LIN {X 0,Y 197.942,Z 460.439,A -85,B 0,C 180,E1 -21324.546,E2 -21324.546} C_VEL
LIN {X 0,Y 197.661,Z 463.395,A -85,B 0,C 180,E1 -21327.96,E2 -21327.96} C_VEL
LIN {X 0,Y 197.713,Z 464.596,A -85,B 0,C 180,E1 -21329.998,E2 -21329.998} C_VEL
LIN {X 0,Y 197.549,Z 465.339,A -85,B 0,C 180,E1 -21332.037,E2 -21332.037} C_VEL
LIN {X 0,Y 197.391,Z 465.599,A -85,B 0,C 180,E1 -21336.129,E2 -21336.129} C_VEL
LIN {X 0,Y 197.553,Z 465.155,A -85,B 0,C 180,E1 -21338.179,E2 -21338.179} C_VEL
LIN {X 0,Y 197.931,Z 464.289,A -85,B 0,C 180,E1 -21340.224,E2 -21340.224} C_VEL
LIN {X 0,Y 199.286,Z 461.345,A -85,B 0,C 180,E1 -21344.29,E2 -21344.29} C_VEL
LIN {X 0,Y 201.111,Z 458.021,A -85,B 0,C 180,E1 -21347.278,E2 -21347.278} C_VEL
LIN {X 0,Y 203.402,Z 453.64,A -85,B 0,C 180,E1 -21350.211,E2 -21350.211} C_VEL
LIN {X 0,Y 206.215,Z 447.922,A -85,B 0,C 180,E1 -21353.155,E2 -21353.155} C_VEL
LIN {X 0,Y 209.5,Z 441.158,A -85,B 0,C 180,E1 -21355.853,E2 -21355.853} C_VEL
LIN {X 0,Y 213.512,Z 432.506,A -85,B 0,C 180,E1 -21358.506,E2 -21358.506} C_VEL
LIN {X 0,Y 217.222,Z 423.657,A -85,B 0,C 180,E1 -21360.633,E2 -21360.633} C_VEL
LIN {X 0,Y 220.793,Z 413.95,A -85,B 0,C 180,E1 -21362.487,E2 -21362.487} C_VEL
LIN {X 0,Y 224.184,Z 403.229,A -85,B 0,C 180,E1 -21364.079,E2 -21364.079} C_VEL
LIN {X 0,Y 227.453,Z 391.24,A -85,B 0,C 180,E1 -21365.402,E2 -21365.402} C_VEL
LIN {X 0,Y 230.075,Z 378.731,A -85,B 0,C 180,E1 -21366.421,E2 -21366.421} C_VEL
LIN {X 0,Y 231.955,Z 365.313,A -85,B 0,C 180,E1 -21367.16,E2 -21367.16} C_VEL
LIN {X 0,Y 233.15,Z 348.218,A -85,B 0,C 180,E1 -21367.736,E2 -21367.736} C_VEL
LIN {X 0,Y 234.841,Z 317.353,A -85,B 0,C 180,E1 -21368.645,E2 -21368.645} C_VEL
LIN {X 0,Y 232.576,Z 295.848,A -85,B 0,C 180,E1 -21370.122,E2 -21370.122} C_VEL
LIN {X 0,Y 230.05,Z 288.532,A -85,B 0,C 180,E1 -21371.098,E2 -21371.098} C_VEL
LIN {X 0,Y 224.045,Z 278.534,A -85,B 0,C 180,E1 -21373.235,E2 -21373.235} C_VEL
LIN {X 0,Y 217.477,Z 268.652,A -85,B 0,C 180,E1 -21375.773,E2 -21375.773} C_VEL
LIN {X 0,Y 213.24,Z 263.042,A -85,B 0,C 180,E1 -21377.545,E2 -21377.545} C_VEL
LIN {X 0,Y 210.962,Z 259.841,A -85,B 0,C 180,E1 -21378.571,E2 -21378.571} C_VEL
LIN {X 0,Y 208.26,Z 256.36,A -85,B 0,C 180,E1 -21379.834,E2 -21379.834} C_VEL
LIN {X 0,Y 207.427,Z 255.193,A -85,B 0,C 180,E1 -21380.244,E2 -21380.244} C_VEL
LIN {X 0,Y 204.921,Z 252.53,A -85,B 0,C 180,E1 -21381.473,E2 -21381.473} C_VEL
LIN {X 0,Y 203.6,Z 250.132,A -85,B 0,C 180,E1 -21382.215,E2 -21382.215} C_VEL
LIN {X 0,Y 201.149,Z 248.227,A -85,B 0,C 180,E1 -21383.488,E2 -21383.488} C_VEL
LIN {X 0,Y 199.87,Z 245.754,A -85,B 0,C 180,E1 -21384.296,E2 -21384.296} C_VEL
LIN {X 0,Y 199.655,Z 244.583,A -85,B 0,C 180,E1 -21384.529,E2 -21384.529} C_VEL
LIN {X 0,Y 199.678,Z 244.597,A -85,B 0,C 180,E1 -21388.133,E2 -21388.133} C_VEL
LIN {X 0,Y 199.633,Z 244.592,A -85,B 0,C 180,E1 -21392.764,E2 -21392.764} C_VEL
LIN {X 0,Y 199.67,Z 244.569,A -85,B 0,C 180,E1 -21397.221,E2 -21397.221} C_VEL
LIN {X 0,Y 199.737,Z 244.601,A -85,B 0,C 180,E1 -21401.802,E2 -21401.802} C_VEL
LIN {X 0,Y 199.795,Z 244.552,A -85,B 0,C 180,E1 -21405.746,E2 -21405.746} C_VEL
LIN {X 0,Y 200.015,Z 244.57,A -85,B 0,C 180,E1 -21409.882,E2 -21409.882} C_VEL
LIN {X 0,Y 199.994,Z 244.528,A -85,B 0,C 180,E1 -21413.949,E2 -21413.949} C_VEL
LIN {X 0,Y 200.281,Z 244.53,A -85,B 0,C 180,E1 -21417.99,E2 -21417.99} C_VEL
LIN {X 0,Y 200.44,Z 244.499,A -85,B 0,C 180,E1 -21420,E2 -21420} C_VEL
LIN {X 0,Y 199.992,Z 244.532,A -85,B 0,C 180,E1 -21424.031,E2 -21424.031} C_VEL
LIN {X 0,Y 200.081,Z 244.539,A -85,B 0,C 180,E1 -21428.077,E2 -21428.077} C_VEL
LIN {X 0,Y 199.863,Z 244.559,A -85,B 0,C 180,E1 -21432.181,E2 -21432.181} C_VEL
LIN {X 0,Y 199.782,Z 244.569,A -85,B 0,C 180,E1 -21436.346,E2 -21436.346} C_VEL
LIN {X 0,Y 199.691,Z 244.611,A -85,B 0,C 180,E1 -21440.607,E2 -21440.607} C_VEL
LIN {X 0,Y 199.718,Z 244.604,A -85,B 0,C 180,E1 -21441.956,E2 -21441.956} C_VEL
LIN {X 0,Y 200.527,Z 247.136,A -85,B 0,C 180,E1 -21442.541,E2 -21442.541} C_VEL
LIN {X 0,Y 202.565,Z 249.424,A -85,B 0,C 180,E1 -21443.668,E2 -21443.668} C_VEL
LIN {X 0,Y 203.976,Z 250.475,A -85,B 0,C 180,E1 -21444.381,E2 -21444.381} C_VEL
LIN {X 0,Y 205.845,Z 253.622,A -85,B 0,C 180,E1 -21445.399,E2 -21445.399} C_VEL
LIN {X 0,Y 208.072,Z 255.817,A -85,B 0,C 180,E1 -21446.461,E2 -21446.461} C_VEL
LIN {X 0,Y 210.626,Z 259.382,A -85,B 0,C 180,E1 -21447.678,E2 -21447.678} C_VEL
LIN {X 0,Y 212.048,Z 261.212,A -85,B 0,C 180,E1 -21448.319,E2 -21448.319} C_VEL
LIN {X 0,Y 215.867,Z 266.452,A -85,B 0,C 180,E1 -21449.971,E2 -21449.971} C_VEL
LIN {X 0,Y 221.051,Z 273.806,A -85,B 0,C 180,E1 -21452.044,E2 -21452.044} C_VEL
LIN {X 0,Y 228.397,Z 285.486,A -85,B 0,C 180,E1 -21454.726,E2 -21454.726} C_VEL
LIN {X 0,Y 235.783,Z 298.796,A -85,B 0,C 180,E1 -21457.196,E2 -21457.196} C_VEL
LIN {X 0,Y 236.31,Z 299.86,A -85,B 0,C 180,E1 -21457.367,E2 -21457.367} C_VEL
LIN {X 0,Y 233.51,Z 345.758,A -85,B 0,C 180,E1 -21458.696,E2 -21458.696} C_VEL
LIN {X 0,Y 232.102,Z 359,A -85,B 0,C 180,E1 -21459.385,E2 -21459.385} C_VEL
LIN {X 0,Y 229.988,Z 371.479,A -85,B 0,C 180,E1 -21460.359,E2 -21460.359} C_VEL
LIN {X 0,Y 227.13,Z 384.146,A -85,B 0,C 180,E1 -21461.716,E2 -21461.716} C_VEL
LIN {X 0,Y 223.756,Z 395.932,A -85,B 0,C 180,E1 -21463.423,E2 -21463.423} C_VEL
LIN {X 0,Y 220.104,Z 406.463,A -85,B 0,C 180,E1 -21465.378,E2 -21465.378} C_VEL
LIN {X 0,Y 216.353,Z 415.831,A -85,B 0,C 180,E1 -21467.624,E2 -21467.624} C_VEL
LIN {X 0,Y 212.904,Z 423.462,A -85,B 0,C 180,E1 -21469.935,E2 -21469.935} C_VEL
LIN {X 0,Y 209.261,Z 430.89,A -85,B 0,C 180,E1 -21472.808,E2 -21472.808} C_VEL
LIN {X 0,Y 206.113,Z 436.751,A -85,B 0,C 180,E1 -21475.766,E2 -21475.766} C_VEL
LIN {X 0,Y 203.456,Z 441.257,A -85,B 0,C 180,E1 -21478.795,E2 -21478.795} C_VEL
LIN {X 0,Y 201.95,Z 443.598,A -85,B 0,C 180,E1 -21480.845,E2 -21480.845} C_VEL
LIN {X 0,Y 200.677,Z 445.486,A -85,B 0,C 180,E1 -21482.92,E2 -21482.92} C_VEL
LIN {X 0,Y 198.945,Z 447.673,A -85,B 0,C 180,E1 -21486.707,E2 -21486.707} C_VEL
LIN {X 0,Y 198.092,Z 448.373,A -85,B 0,C 180,E1 -21489.222,E2 -21489.222} C_VEL
LIN {X 0,Y 197.64,Z 448.461,A -85,B 0,C 180,E1 -21491.337,E2 -21491.337} C_VEL
LIN {X 0,Y 197.323,Z 447.972,A -85,B 0,C 180,E1 -21494.084,E2 -21494.084} C_VEL
LIN {X 0,Y 197.162,Z 446.247,A -85,B 0,C 180,E1 -21497.653,E2 -21497.653} C_VEL
LIN {X 0,Y 197.432,Z 443.697,A -85,B 0,C 180,E1 -21500.785,E2 -21500.785} C_VEL
LIN {X 0,Y 198.046,Z 440.117,A -85,B 0,C 180,E1 -21503.891,E2 -21503.891} C_VEL
LIN {X 0,Y 198.809,Z 435.436,A -85,B 0,C 180,E1 -21506.963,E2 -21506.963} C_VEL
LIN {X 0,Y 199.937,Z 429.504,A -85,B 0,C 180,E1 -21510.002,E2 -21510.002} C_VEL
LIN {X 0,Y 201.503,Z 422.11,A -85,B 0,C 180,E1 -21513.001,E2 -21513.001} C_VEL
LIN {X 0,Y 203.143,Z 414.552,A -85,B 0,C 180,E1 -21515.462,E2 -21515.462} C_VEL
LIN {X 0,Y 205.28,Z 404.301,A -85,B 0,C 180,E1 -21518.121,E2 -21518.121} C_VEL
LIN {X 0,Y 207.44,Z 393.458,A -85,B 0,C 180,E1 -21520.33,E2 -21520.33} C_VEL
LIN {X 0,Y 209.325,Z 382.204,A -85,B 0,C 180,E1 -21522.115,E2 -21522.115} C_VEL
LIN {X 0,Y 210.819,Z 369.938,A -85,B 0,C 180,E1 -21523.62,E2 -21523.62} C_VEL
LIN {X 0,Y 212.169,Z 357.731,A -85,B 0,C 180,E1 -21524.693,E2 -21524.693} C_VEL
LIN {X 0,Y 213.122,Z 344.661,A -85,B 0,C 180,E1 -21525.447,E2 -21525.447} C_VEL
LIN {X 0,Y 215.625,Z 279.151,A -85,B 0,C 180,E1 -21527.583,E2 -21527.583} C_VEL
LIN {X 0,Y 208.838,Z 263.06,A -85,B 0,C 180,E1 -21529.128,E2 -21529.128} C_VEL
LIN {X 0,Y 201.032,Z 247.936,A -85,B 0,C 180,E1 -21530.917,E2 -21530.917} C_VEL
LIN {X 0,Y 199.755,Z 244.973,A -85,B 0,C 180,E1 -21531.246,E2 -21531.246} C_VEL
LIN {X 0,Y 199.699,Z 244.61,A -85,B 0,C 180,E1 -21531.317,E2 -21531.317} C_VEL
LIN {X 0,Y 199.647,Z 244.616,A -85,B 0,C 180,E1 -21534.99,E2 -21534.99} C_VEL
LIN {X 0,Y 199.613,Z 244.619,A -85,B 0,C 180,E1 -21539.535,E2 -21539.535} C_VEL
LIN {X 0,Y 199.671,Z 244.612,A -85,B 0,C 180,E1 -21542.354,E2 -21542.354} C_VEL
LIN {X 0,Y 199.623,Z 244.611,A -85,B 0,C 180,E1 -21546.766,E2 -21546.766} C_VEL
LIN {X 0,Y 199.601,Z 244.623,A -85,B 0,C 180,E1 -21549.333,E2 -21549.333} C_VEL
LIN {X 0,Y 199.572,Z 244.612,A -85,B 0,C 180,E1 -21552.308,E2 -21552.308} C_VEL
LIN {X 0,Y 199.582,Z 244.619,A -85,B 0,C 180,E1 -21555.228,E2 -21555.228} C_VEL
LIN {X 0,Y 199.575,Z 244.621,A -85,B 0,C 180,E1 -21558.003,E2 -21558.003} C_VEL
LIN {X 0,Y 199.602,Z 244.602,A -85,B 0,C 180,E1 -21560.774,E2 -21560.774} C_VEL
LIN {X 0,Y 199.617,Z 244.617,A -85,B 0,C 180,E1 -21565.714,E2 -21565.714} C_VEL
LIN {X 0,Y 199.692,Z 244.605,A -85,B 0,C 180,E1 -21568.135,E2 -21568.135} C_VEL
LIN {X 0,Y 199.734,Z 244.589,A -85,B 0,C 180,E1 -21572.188,E2 -21572.188} C_VEL
LIN {X 0,Y 206.813,Z 272.195,A -85,B 0,C 180,E1 -21574.133,E2 -21574.133} C_VEL
LIN {X 0,Y 203.31,Z 347.013,A -85,B 0,C 180,E1 -21578.76,E2 -21578.76} C_VEL
LIN {X 0,Y 202.562,Z 361.775,A -85,B 0,C 180,E1 -21580.095,E2 -21580.095} C_VEL
LIN {X 0,Y 201.607,Z 374.93,A -85,B 0,C 180,E1 -21581.715,E2 -21581.715} C_VEL
LIN {X 0,Y 200.603,Z 387.656,A -85,B 0,C 180,E1 -21583.723,E2 -21583.723} C_VEL
LIN {X 0,Y 199.784,Z 399.17,A -85,B 0,C 180,E1 -21586.004,E2 -21586.004} C_VEL
LIN {X 0,Y 199.015,Z 408.647,A -85,B 0,C 180,E1 -21588.284,E2 -21588.284} C_VEL
LIN {X 0,Y 198.445,Z 417.441,A -85,B 0,C 180,E1 -21590.829,E2 -21590.829} C_VEL
LIN {X 0,Y 198.005,Z 426.054,A -85,B 0,C 180,E1 -21593.887,E2 -21593.887} C_VEL
LIN {X 0,Y 197.786,Z 433.046,A -85,B 0,C 180,E1 -21596.944,E2 -21596.944} C_VEL
LIN {X 0,Y 197.683,Z 438.659,A -85,B 0,C 180,E1 -21600,E2 -21600} C_VEL
LIN {X 0,Y 197.968,Z 443.125,A -85,B 0,C 180,E1 -21603.052,E2 -21603.052} C_VEL
LIN {X 0,Y 198.708,Z 446.59,A -85,B 0,C 180,E1 -21606.09,E2 -21606.09} C_VEL
LIN {X 0,Y 200.084,Z 449.8,A -85,B 0,C 180,E1 -21610.115,E2 -21610.115} C_VEL
LIN {X 0,Y 201.178,Z 450.837,A -85,B 0,C 180,E1 -21612.099,E2 -21612.099} C_VEL
LIN {X 0,Y 204.584,Z 451.772,A -85,B 0,C 180,E1 -21615.951,E2 -21615.951} C_VEL
LIN {X 0,Y 208.896,Z 451.263,A -85,B 0,C 180,E1 -21619.659,E2 -21619.659} C_VEL
LIN {X 0,Y 214.052,Z 449.305,A -85,B 0,C 180,E1 -21623.203,E2 -21623.203} C_VEL
LIN {X 0,Y 220.272,Z 445.773,A -85,B 0,C 180,E1 -21626.531,E2 -21626.531} C_VEL
LIN {X 0,Y 224.069,Z 443.144,A -85,B 0,C 180,E1 -21628.292,E2 -21628.292} C_VEL
LIN {X 0,Y 226.413,Z 441.172,A -85,B 0,C 180,E1 -21629.578,E2 -21629.578} C_VEL
LIN {X 0,Y 231.508,Z 435.44,A -85,B 0,C 180,E1 -21633.602,E2 -21633.602} C_VEL
LIN {X 0,Y 233.945,Z 432.914,A -85,B 0,C 180,E1 -21634.759,E2 -21634.759} C_VEL
LIN {X 0,Y 234.952,Z 431.935,A -85,B 0,C 180,E1 -21635.093,E2 -21635.093} C_VEL
LIN {X 0,Y 243.29,Z 423.495,A -85,B 0,C 180,E1 -21637.346,E2 -21637.346} C_VEL
LIN {X 0,Y 250.623,Z 414.818,A -85,B 0,C 180,E1 -21639.12,E2 -21639.12} C_VEL
LIN {X 0,Y 258.387,Z 404.268,A -85,B 0,C 180,E1 -21640.752,E2 -21640.752} C_VEL
LIN {X 0,Y 265.576,Z 392.717,A -85,B 0,C 180,E1 -21642.106,E2 -21642.106} C_VEL
LIN {X 0,Y 271.928,Z 380.59,A -85,B 0,C 180,E1 -21643.21,E2 -21643.21} C_VEL
LIN {X 0,Y 276.977,Z 368.919,A -85,B 0,C 180,E1 -21643.996,E2 -21643.996} C_VEL
LIN {X 0,Y 276.871,Z 369.239,A -85,B 0,C 180,E1 -21644.215,E2 -21644.215} C_VEL
LIN {X 0,Y 271.282,Z 382.338,A -85,B 0,C 180,E1 -21644.913,E2 -21644.913} C_VEL
LIN {X 0,Y 264.304,Z 395.717,A -85,B 0,C 180,E1 -21645.885,E2 -21645.885} C_VEL
LIN {X 0,Y 256.722,Z 407.968,A -85,B 0,C 180,E1 -21647.078,E2 -21647.078} C_VEL
LIN {X 0,Y 249.17,Z 418.536,A -85,B 0,C 180,E1 -21648.482,E2 -21648.482} C_VEL
LIN {X 0,Y 241.34,Z 428.187,A -85,B 0,C 180,E1 -21650.157,E2 -21650.157} C_VEL
LIN {X 0,Y 233.944,Z 436.234,A -85,B 0,C 180,E1 -21651.984,E2 -21651.984} C_VEL
LIN {X 0,Y 227.076,Z 442.972,A -85,B 0,C 180,E1 -21653.979,E2 -21653.979} C_VEL
LIN {X 0,Y 218.693,Z 450.246,A -85,B 0,C 180,E1 -21656.883,E2 -21656.883} C_VEL
LIN {X 0,Y 212.811,Z 454.741,A -85,B 0,C 180,E1 -21659.343,E2 -21659.343} C_VEL
LIN {X 0,Y 207.842,Z 458.064,A -85,B 0,C 180,E1 -21661.743,E2 -21661.743} C_VEL
LIN {X 0,Y 202.079,Z 461.387,A -85,B 0,C 180,E1 -21665.331,E2 -21665.331} C_VEL
LIN {X 0,Y 197.481,Z 463.356,A -85,B 0,C 180,E1 -21669.15,E2 -21669.15} C_VEL
LIN {X 0,Y 193.954,Z 463.965,A -85,B 0,C 180,E1 -21673.147,E2 -21673.147} C_VEL
LIN {X 0,Y 191.876,Z 463.198,A -85,B 0,C 180,E1 -21677.302,E2 -21677.302} C_VEL
LIN {X 0,Y 191.007,Z 461.056,A -85,B 0,C 180,E1 -21681.534,E2 -21681.534} C_VEL
LIN {X 0,Y 191.007,Z 459.364,A -85,B 0,C 180,E1 -21683.798,E2 -21683.798} C_VEL
LIN {X 0,Y 190.663,Z 461.301,A -85,B 0,C 180,E1 -21685.77,E2 -21685.77} C_VEL
LIN {X 0,Y 190.578,Z 462.945,A -85,B 0,C 180,E1 -21687.884,E2 -21687.884} C_VEL
LIN {X 0,Y 190.642,Z 464.177,A -85,B 0,C 180,E1 -21689.998,E2 -21689.998} C_VEL
LIN {X 0,Y 190.457,Z 464.976,A -85,B 0,C 180,E1 -21692.112,E2 -21692.112} C_VEL
LIN {X 0,Y 190.301,Z 465.336,A -85,B 0,C 180,E1 -21694.341,E2 -21694.341} C_VEL
LIN {X 0,Y 190.502,Z 464.884,A -85,B 0,C 180,E1 -21698.484,E2 -21698.484} C_VEL
LIN {X 0,Y 190.931,Z 464.077,A -85,B 0,C 180,E1 -21700.603,E2 -21700.603} C_VEL
LIN {X 0,Y 192.377,Z 461.198,A -85,B 0,C 180,E1 -21704.814,E2 -21704.814} C_VEL
LIN {X 0,Y 194.324,Z 457.944,A -85,B 0,C 180,E1 -21707.901,E2 -21707.901} C_VEL
LIN {X 0,Y 196.747,Z 453.637,A -85,B 0,C 180,E1 -21710.926,E2 -21710.926} C_VEL
LIN {X 0,Y 200.096,Z 447.25,A -85,B 0,C 180,E1 -21714.317,E2 -21714.317} C_VEL
LIN {X 0,Y 203.791,Z 440.034,A -85,B 0,C 180,E1 -21717.187,E2 -21717.187} C_VEL
LIN {X 0,Y 208.073,Z 431.218,A -85,B 0,C 180,E1 -21719.879,E2 -21719.879} C_VEL
LIN {X 0,Y 211.955,Z 422.179,A -85,B 0,C 180,E1 -21722.038,E2 -21722.038} C_VEL
LIN {X 0,Y 215.67,Z 412.151,A -85,B 0,C 180,E1 -21723.918,E2 -21723.918} C_VEL
LIN {X 0,Y 219.306,Z 401.05,A -85,B 0,C 180,E1 -21725.507,E2 -21725.507} C_VEL
LIN {X 0,Y 222.249,Z 390.529,A -85,B 0,C 180,E1 -21726.643,E2 -21726.643} C_VEL
LIN {X 0,Y 224.954,Z 377.839,A -85,B 0,C 180,E1 -21727.671,E2 -21727.671} C_VEL
LIN {X 0,Y 226.877,Z 364.287,A -85,B 0,C 180,E1 -21728.413,E2 -21728.413} C_VEL
LIN {X 0,Y 228.259,Z 344.643,A -85,B 0,C 180,E1 -21729.054,E2 -21729.054} C_VEL
LIN {X 0,Y 229.726,Z 318.386,A -85,B 0,C 180,E1 -21729.845,E2 -21729.845} C_VEL
LIN {X 0,Y 227.794,Z 298.718,A -85,B 0,C 180,E1 -21731.234,E2 -21731.234} C_VEL
LIN {X 0,Y 225.766,Z 292.778,A -85,B 0,C 180,E1 -21732.064,E2 -21732.064} C_VEL
LIN {X 0,Y 219.255,Z 281.77,A -85,B 0,C 180,E1 -21734.522,E2 -21734.522} C_VEL
LIN {X 0,Y 212.694,Z 272.179,A -85,B 0,C 180,E1 -21737.234,E2 -21737.234} C_VEL
LIN {X 0,Y 208.014,Z 265.668,A -85,B 0,C 180,E1 -21739.374,E2 -21739.374} C_VEL
LIN {X 0,Y 204.614,Z 261.189,A -85,B 0,C 180,E1 -21741.054,E2 -21741.054} C_VEL
LIN {X 0,Y 201.939,Z 257.971,A -85,B 0,C 180,E1 -21742.453,E2 -21742.453} C_VEL
LIN {X 0,Y 200.884,Z 256.326,A -85,B 0,C 180,E1 -21743.057,E2 -21743.057} C_VEL
LIN {X 0,Y 198.394,Z 253.892,A -85,B 0,C 180,E1 -21744.452,E2 -21744.452} C_VEL
LIN {X 0,Y 196.839,Z 251.132,A -85,B 0,C 180,E1 -21745.473,E2 -21745.473} C_VEL
LIN {X 0,Y 194.32,Z 249.334,A -85,B 0,C 180,E1 -21747.021,E2 -21747.021} C_VEL
LIN {X 0,Y 192.972,Z 246.91,A -85,B 0,C 180,E1 -21748.025,E2 -21748.025} C_VEL
LIN {X 0,Y 192.605,Z 245.47,A -85,B 0,C 180,E1 -21748.44,E2 -21748.44} C_VEL
LIN {X 0,Y 192.611,Z 245.454,A -85,B 0,C 180,E1 -21751.684,E2 -21751.684} C_VEL
LIN {X 0,Y 192.662,Z 245.449,A -85,B 0,C 180,E1 -21756.343,E2 -21756.343} C_VEL
LIN {X 0,Y 192.686,Z 245.477,A -85,B 0,C 180,E1 -21761.491,E2 -21761.491} C_VEL
LIN {X 0,Y 192.721,Z 245.435,A -85,B 0,C 180,E1 -21765.211,E2 -21765.211} C_VEL
LIN {X 0,Y 192.937,Z 245.447,A -85,B 0,C 180,E1 -21769.567,E2 -21769.567} C_VEL
LIN {X 0,Y 192.958,Z 245.405,A -85,B 0,C 180,E1 -21773.727,E2 -21773.727} C_VEL
LIN {X 0,Y 193.225,Z 245.406,A -85,B 0,C 180,E1 -21777.916,E2 -21777.916} C_VEL
LIN {X 0,Y 193.406,Z 245.373,A -85,B 0,C 180,E1 -21780,E2 -21780} C_VEL
LIN {X 0,Y 192.939,Z 245.411,A -85,B 0,C 180,E1 -21784.178,E2 -21784.178} C_VEL
LIN {X 0,Y 193.029,Z 245.412,A -85,B 0,C 180,E1 -21788.375,E2 -21788.375} C_VEL
LIN {X 0,Y 192.79,Z 245.445,A -85,B 0,C 180,E1 -21792.635,E2 -21792.635} C_VEL
LIN {X 0,Y 192.77,Z 245.63,A -85,B 0,C 180,E1 -21798.151,E2 -21798.151} C_VEL
LIN {X 0,Y 193.576,Z 248.103,A -85,B 0,C 180,E1 -21798.85,E2 -21798.85} C_VEL
LIN {X 0,Y 195.45,Z 250.299,A -85,B 0,C 180,E1 -21800.112,E2 -21800.112} C_VEL
LIN {X 0,Y 197.285,Z 251.592,A -85,B 0,C 180,E1 -21801.212,E2 -21801.212} C_VEL
LIN {X 0,Y 199.104,Z 254.644,A -85,B 0,C 180,E1 -21802.369,E2 -21802.369} C_VEL
LIN {X 0,Y 201.519,Z 256.996,A -85,B 0,C 180,E1 -21803.692,E2 -21803.692} C_VEL
LIN {X 0,Y 203.924,Z 260.43,A -85,B 0,C 180,E1 -21805.003,E2 -21805.003} C_VEL
LIN {X 0,Y 205.433,Z 262.08,A -85,B 0,C 180,E1 -21805.755,E2 -21805.755} C_VEL
LIN {X 0,Y 208.337,Z 265.837,A -85,B 0,C 180,E1 -21807.168,E2 -21807.168} C_VEL
LIN {X 0,Y 214.92,Z 275.173,A -85,B 0,C 180,E1 -21810.117,E2 -21810.117} C_VEL
LIN {X 0,Y 220.68,Z 284.054,A -85,B 0,C 180,E1 -21812.441,E2 -21812.441} C_VEL
LIN {X 0,Y 226.778,Z 294.388,A -85,B 0,C 180,E1 -21814.695,E2 -21814.695} C_VEL
LIN {X 0,Y 231.073,Z 302.377,A -85,B 0,C 180,E1 -21816.191,E2 -21816.191} C_VEL
LIN {X 0,Y 228.288,Z 346.944,A -85,B 0,C 180,E1 -21817.522,E2 -21817.522} C_VEL
LIN {X 0,Y 226.836,Z 359.727,A -85,B 0,C 180,E1 -21818.216,E2 -21818.216} C_VEL
LIN {X 0,Y 224.549,Z 372.481,A -85,B 0,C 180,E1 -21819.232,E2 -21819.232} C_VEL
LIN {X 0,Y 221.809,Z 384.128,A -85,B 0,C 180,E1 -21820.501,E2 -21820.501} C_VEL
LIN {X 0,Y 218.279,Z 395.995,A -85,B 0,C 180,E1 -21822.226,E2 -21822.226} C_VEL
LIN {X 0,Y 214.488,Z 406.574,A -85,B 0,C 180,E1 -21824.215,E2 -21824.215} C_VEL
LIN {X 0,Y 210.905,Z 415.151,A -85,B 0,C 180,E1 -21826.258,E2 -21826.258} C_VEL
LIN {X 0,Y 207.114,Z 423.272,A -85,B 0,C 180,E1 -21828.72,E2 -21828.72} C_VEL
LIN {X 0,Y 203.378,Z 430.533,A -85,B 0,C 180,E1 -21831.54,E2 -21831.54} C_VEL
LIN {X 0,Y 199.996,Z 436.543,A -85,B 0,C 180,E1 -21834.565,E2 -21834.565} C_VEL
LIN {X 0,Y 197.116,Z 441.196,A -85,B 0,C 180,E1 -21837.672,E2 -21837.672} C_VEL
LIN {X 0,Y 195.492,Z 443.598,A -85,B 0,C 180,E1 -21839.784,E2 -21839.784} C_VEL
LIN {X 0,Y 194.078,Z 445.539,A -85,B 0,C 180,E1 -21841.919,E2 -21841.919} C_VEL
LIN {X 0,Y 192.933,Z 447.023,A -85,B 0,C 180,E1 -21844.082,E2 -21844.082} C_VEL
LIN {X 0,Y 191.991,Z 448.026,A -85,B 0,C 180,E1 -21846.258,E2 -21846.258} C_VEL
LIN {X 0,Y 191.208,Z 448.624,A -85,B 0,C 180,E1 -21848.437,E2 -21848.437} C_VEL
LIN {X 0,Y 190.667,Z 448.807,A -85,B 0,C 180,E1 -21850.628,E2 -21850.628} C_VEL
LIN {X 0,Y 190.25,Z 448.282,A -85,B 0,C 180,E1 -21853.837,E2 -21853.837} C_VEL
LIN {X 0,Y 190.077,Z 446.773,A -85,B 0,C 180,E1 -21857.185,E2 -21857.185} C_VEL
LIN {X 0,Y 190.17,Z 445.231,A -85,B 0,C 180,E1 -21859.354,E2 -21859.354} C_VEL
LIN {X 0,Y 190.649,Z 442.106,A -85,B 0,C 180,E1 -21862.589,E2 -21862.589} C_VEL
LIN {X 0,Y 191.38,Z 437.915,A -85,B 0,C 180,E1 -21865.79,E2 -21865.79} C_VEL
LIN {X 0,Y 192.596,Z 431.548,A -85,B 0,C 180,E1 -21869.48,E2 -21869.48} C_VEL
LIN {X 0,Y 194.087,Z 424.564,A -85,B 0,C 180,E1 -21872.597,E2 -21872.597} C_VEL
LIN {X 0,Y 196.041,Z 415.829,A -85,B 0,C 180,E1 -21875.66,E2 -21875.66} C_VEL
LIN {X 0,Y 198.026,Z 406.876,A -85,B 0,C 180,E1 -21878.164,E2 -21878.164} C_VEL
LIN {X 0,Y 200.159,Z 396.745,A -85,B 0,C 180,E1 -21880.412,E2 -21880.412} C_VEL
LIN {X 0,Y 202.163,Z 385.992,A -85,B 0,C 180,E1 -21882.296,E2 -21882.296} C_VEL
LIN {X 0,Y 203.651,Z 375.737,A -85,B 0,C 180,E1 -21883.727,E2 -21883.727} C_VEL
LIN {X 0,Y 204.962,Z 364.794,A -85,B 0,C 180,E1 -21884.904,E2 -21884.904} C_VEL
LIN {X 0,Y 206.183,Z 351.773,A -85,B 0,C 180,E1 -21885.893,E2 -21885.893} C_VEL
LIN {X 0,Y 207.057,Z 336.722,A -85,B 0,C 180,E1 -21886.556,E2 -21886.556} C_VEL
LIN {X 0,Y 209.219,Z 280.86,A -85,B 0,C 180,E1 -21888.391,E2 -21888.391} C_VEL
LIN {X 0,Y 202.464,Z 265.01,A -85,B 0,C 180,E1 -21890.002,E2 -21890.002} C_VEL
LIN {X 0,Y 194.005,Z 248.862,A -85,B 0,C 180,E1 -21892.058,E2 -21892.058} C_VEL
LIN {X 0,Y 192.776,Z 246.207,A -85,B 0,C 180,E1 -21892.389,E2 -21892.389} C_VEL
LIN {X 0,Y 192.648,Z 245.484,A -85,B 0,C 180,E1 -21892.526,E2 -21892.526} C_VEL
LIN {X 0,Y 192.625,Z 245.492,A -85,B 0,C 180,E1 -21898.317,E2 -21898.317} C_VEL
LIN {X 0,Y 192.601,Z 245.494,A -85,B 0,C 180,E1 -21903.188,E2 -21903.188} C_VEL
LIN {X 0,Y 192.548,Z 245.5,A -85,B 0,C 180,E1 -21908.355,E2 -21908.355} C_VEL
LIN {X 0,Y 192.49,Z 245.492,A -85,B 0,C 180,E1 -21913.094,E2 -21913.094} C_VEL
LIN {X 0,Y 192.491,Z 245.506,A -85,B 0,C 180,E1 -21916.908,E2 -21916.908} C_VEL
LIN {X 0,Y 192.547,Z 245.478,A -85,B 0,C 180,E1 -21921.646,E2 -21921.646} C_VEL
LIN {X 0,Y 192.602,Z 245.492,A -85,B 0,C 180,E1 -21926.814,E2 -21926.814} C_VEL
LIN {X 0,Y 192.686,Z 245.465,A -85,B 0,C 180,E1 -21931.985,E2 -21931.985} C_VEL
LIN {X 0,Y 199.653,Z 272.654,A -85,B 0,C 180,E1 -21933.961,E2 -21933.961} C_VEL
LIN {X 0,Y 196.212,Z 346.805,A -85,B 0,C 180,E1 -21938.763,E2 -21938.763} C_VEL
LIN {X 0,Y 195.478,Z 361.732,A -85,B 0,C 180,E1 -21940.165,E2 -21940.165} C_VEL
LIN {X 0,Y 194.513,Z 374.883,A -85,B 0,C 180,E1 -21941.842,E2 -21941.842} C_VEL
LIN {X 0,Y 193.493,Z 387.661,A -85,B 0,C 180,E1 -21943.921,E2 -21943.921} C_VEL
LIN {X 0,Y 192.717,Z 399.186,A -85,B 0,C 180,E1 -21946.287,E2 -21946.287} C_VEL
LIN {X 0,Y 191.846,Z 409.612,A -85,B 0,C 180,E1 -21948.911,E2 -21948.911} C_VEL
LIN {X 0,Y 191.319,Z 418.255,A -85,B 0,C 180,E1 -21951.55,E2 -21951.55} C_VEL
LIN {X 0,Y 190.941,Z 425.687,A -85,B 0,C 180,E1 -21954.288,E2 -21954.288} C_VEL
LIN {X 0,Y 190.769,Z 432.588,A -85,B 0,C 180,E1 -21957.36,E2 -21957.36} C_VEL
LIN {X 0,Y 190.707,Z 439.165,A -85,B 0,C 180,E1 -21961.055,E2 -21961.055} C_VEL
LIN {X 0,Y 191.143,Z 443.591,A -85,B 0,C 180,E1 -21964.217,E2 -21964.217} C_VEL
LIN {X 0,Y 191.686,Z 446.011,A -85,B 0,C 180,E1 -21966.314,E2 -21966.314} C_VEL
LIN {X 0,Y 192.334,Z 447.987,A -85,B 0,C 180,E1 -21968.404,E2 -21968.404} C_VEL
LIN {X 0,Y 194.253,Z 450.787,A -85,B 0,C 180,E1 -21972.537,E2 -21972.537} C_VEL
LIN {X 0,Y 197.78,Z 452.167,A -85,B 0,C 180,E1 -21976.515,E2 -21976.515} C_VEL
LIN {X 0,Y 202.272,Z 452.089,A -85,B 0,C 180,E1 -21980.331,E2 -21980.331} C_VEL
LIN {X 0,Y 207.659,Z 450.555,A -85,B 0,C 180,E1 -21983.961,E2 -21983.961} C_VEL
LIN {X 0,Y 214.14,Z 447.555,A -85,B 0,C 180,E1 -21987.353,E2 -21987.353} C_VEL
LIN {X 0,Y 219.521,Z 444.285,A -85,B 0,C 180,E1 -21989.751,E2 -21989.751} C_VEL
LIN {X 0,Y 225.44,Z 440.066,A -85,B 0,C 180,E1 -21992.003,E2 -21992.003} C_VEL
LIN {X 0,Y 231.749,Z 434.856,A -85,B 0,C 180,E1 -21994.127,E2 -21994.127} C_VEL
LIN {X 0,Y 234.952,Z 431.935,A -85,B 0,C 180,E1 -21995.093,E2 -21995.093} C_VEL
LIN {X 0,Y 237.823,Z 429.073,A -85,B 0,C 180,E1 -21996.141,E2 -21996.141} C_VEL
LIN {X 0,Y 244.81,Z 420.956,A -85,B 0,C 180,E1 -21999.522,E2 -21999.522} C_VEL
LIN {X 0,Y 247.589,Z 417.583,A -85,B 0,C 180,E1 -22000.431,E2 -22000.431} C_VEL
LIN {X 0,Y 248.636,Z 416.318,A -85,B 0,C 180,E1 -22000.676,E2 -22000.676} C_VEL
LIN {X 0,Y 256.389,Z 406.474,A -85,B 0,C 180,E1 -22002.188,E2 -22002.188} C_VEL
LIN {X 0,Y 264.046,Z 395.095,A -85,B 0,C 180,E1 -22003.51,E2 -22003.51} C_VEL
LIN {X 0,Y 264.82,Z 393.816,A -85,B 0,C 180,E1 -22003.631,E2 -22003.631} C_VEL
LIN {X 0,Y 265.833,Z 392.182,A -85,B 0,C 180,E1 -22004.032,E2 -22004.032} C_VEL
LIN {X 0,Y 258.502,Z 403.99,A -85,B 0,C 180,E1 -22005.017,E2 -22005.017} C_VEL
LIN {X 0,Y 251.189,Z 414.213,A -85,B 0,C 180,E1 -22006.171,E2 -22006.171} C_VEL
LIN {X 0,Y 242.808,Z 424.421,A -85,B 0,C 180,E1 -22007.701,E2 -22007.701} C_VEL
LIN {X 0,Y 233.573,Z 434.218,A -85,B 0,C 180,E1 -22009.688,E2 -22009.688} C_VEL
LIN {X 0,Y 225.029,Z 442.185,A -85,B 0,C 180,E1 -22011.913,E2 -22011.913} C_VEL
LIN {X 0,Y 217.093,Z 448.648,A -85,B 0,C 180,E1 -22014.356,E2 -22014.356} C_VEL
LIN {X 0,Y 208.929,Z 454.454,A -85,B 0,C 180,E1 -22017.436,E2 -22017.436} C_VEL
LIN {X 0,Y 201.667,Z 458.759,A -85,B 0,C 180,E1 -22020.795,E2 -22020.795} C_VEL
LIN {X 0,Y 195.653,Z 461.606,A -85,B 0,C 180,E1 -22024.463,E2 -22024.463} C_VEL
LIN {X 0,Y 190.851,Z 463.132,A -85,B 0,C 180,E1 -22028.39,E2 -22028.39} C_VEL
LIN {X 0,Y 187.176,Z 463.337,A -85,B 0,C 180,E1 -22032.517,E2 -22032.517} C_VEL
LIN {X 0,Y 185.003,Z 462.246,A -85,B 0,C 180,E1 -22036.822,E2 -22036.822} C_VEL
LIN {X 0,Y 184.076,Z 459.773,A -85,B 0,C 180,E1 -22041.213,E2 -22041.213} C_VEL
LIN {X 0,Y 184.043,Z 458.351,A -85,B 0,C 180,E1 -22043.144,E2 -22043.144} C_VEL
LIN {X 0,Y 183.589,Z 460.818,A -85,B 0,C 180,E1 -22045.607,E2 -22045.607} C_VEL
LIN {X 0,Y 183.499,Z 462.494,A -85,B 0,C 180,E1 -22047.803,E2 -22047.803} C_VEL
LIN {X 0,Y 183.572,Z 463.758,A -85,B 0,C 180,E1 -22049.998,E2 -22049.998} C_VEL
LIN {X 0,Y 183.368,Z 464.597,A -85,B 0,C 180,E1 -22052.194,E2 -22052.194} C_VEL
LIN {X 0,Y 183.226,Z 465,A -85,B 0,C 180,E1 -22054.397,E2 -22054.397} C_VEL
LIN {X 0,Y 183.473,Z 464.614,A -85,B 0,C 180,E1 -22058.811,E2 -22058.811} C_VEL
LIN {X 0,Y 183.919,Z 463.851,A -85,B 0,C 180,E1 -22061.012,E2 -22061.012} C_VEL
LIN {X 0,Y 184.6,Z 462.661,A -85,B 0,C 180,E1 -22063.202,E2 -22063.202} C_VEL
LIN {X 0,Y 186.124,Z 460.125,A -85,B 0,C 180,E1 -22066.449,E2 -22066.449} C_VEL
LIN {X 0,Y 188.326,Z 456.604,A -85,B 0,C 180,E1 -22069.622,E2 -22069.622} C_VEL
LIN {X 0,Y 191.112,Z 451.995,A -85,B 0,C 180,E1 -22072.711,E2 -22072.711} C_VEL
LIN {X 0,Y 194.284,Z 446.162,A -85,B 0,C 180,E1 -22075.724,E2 -22075.724} C_VEL
LIN {X 0,Y 198.23,Z 438.906,A -85,B 0,C 180,E1 -22078.593,E2 -22078.593} C_VEL
LIN {X 0,Y 202.731,Z 429.927,A -85,B 0,C 180,E1 -22081.33,E2 -22081.33} C_VEL
LIN {X 0,Y 207.254,Z 419.561,A -85,B 0,C 180,E1 -22083.727,E2 -22083.727} C_VEL
LIN {X 0,Y 211.217,Z 409.043,A -85,B 0,C 180,E1 -22085.609,E2 -22085.609} C_VEL
LIN {X 0,Y 214.584,Z 398.871,A -85,B 0,C 180,E1 -22086.997,E2 -22086.997} C_VEL
LIN {X 0,Y 217.924,Z 386.7,A -85,B 0,C 180,E1 -22088.225,E2 -22088.225} C_VEL
LIN {X 0,Y 220.452,Z 374.051,A -85,B 0,C 180,E1 -22089.167,E2 -22089.167} C_VEL
LIN {X 0,Y 222.135,Z 361.4,A -85,B 0,C 180,E1 -22089.796,E2 -22089.796} C_VEL
LIN {X 0,Y 224.764,Z 319.695,A -85,B 0,C 180,E1 -22091.082,E2 -22091.082} C_VEL
LIN {X 0,Y 223.076,Z 301.559,A -85,B 0,C 180,E1 -22092.405,E2 -22092.405} C_VEL
LIN {X 0,Y 221.681,Z 297.243,A -85,B 0,C 180,E1 -22093.017,E2 -22093.017} C_VEL
LIN {X 0,Y 215.508,Z 286.687,A -85,B 0,C 180,E1 -22095.473,E2 -22095.473} C_VEL
LIN {X 0,Y 208.345,Z 275.892,A -85,B 0,C 180,E1 -22098.641,E2 -22098.641} C_VEL
LIN {X 0,Y 204.631,Z 270.888,A -85,B 0,C 180,E1 -22100.438,E2 -22100.438} C_VEL
LIN {X 0,Y 201.807,Z 267.089,A -85,B 0,C 180,E1 -22101.909,E2 -22101.909} C_VEL
LIN {X 0,Y 199.037,Z 263.426,A -85,B 0,C 180,E1 -22103.453,E2 -22103.453} C_VEL
LIN {X 0,Y 197.84,Z 262.067,A -85,B 0,C 180,E1 -22104.14,E2 -22104.14} C_VEL
LIN {X 0,Y 195.393,Z 259.018,A -85,B 0,C 180,E1 -22105.65,E2 -22105.65} C_VEL
LIN {X 0,Y 194.516,Z 257.582,A -85,B 0,C 180,E1 -22106.247,E2 -22106.247} C_VEL
LIN {X 0,Y 191.991,Z 255.376,A -85,B 0,C 180,E1 -22107.906,E2 -22107.906} C_VEL
LIN {X 0,Y 190.222,Z 252.167,A -85,B 0,C 180,E1 -22109.315,E2 -22109.315} C_VEL
LIN {X 0,Y 187.594,Z 250.491,A -85,B 0,C 180,E1 -22111.313,E2 -22111.313} C_VEL
LIN {X 0,Y 185.91,Z 248.001,A -85,B 0,C 180,E1 -22112.871,E2 -22112.871} C_VEL
LIN {X 0,Y 185.522,Z 246.358,A -85,B 0,C 180,E1 -22113.418,E2 -22113.418} C_VEL
LIN {X 0,Y 185.545,Z 246.325,A -85,B 0,C 180,E1 -22117.743,E2 -22117.743} C_VEL
LIN {X 0,Y 185.642,Z 246.356,A -85,B 0,C 180,E1 -22122.371,E2 -22122.371} C_VEL
LIN {X 0,Y 185.704,Z 246.307,A -85,B 0,C 180,E1 -22126.876,E2 -22126.876} C_VEL
LIN {X 0,Y 185.965,Z 246.311,A -85,B 0,C 180,E1 -22131.306,E2 -22131.306} C_VEL
LIN {X 0,Y 186.171,Z 246.282,A -85,B 0,C 180,E1 -22137.837,E2 -22137.837} C_VEL
LIN {X 0,Y 186.372,Z 246.248,A -85,B 0,C 180,E1 -22140.001,E2 -22140.001} C_VEL
LIN {X 0,Y 185.887,Z 246.29,A -85,B 0,C 180,E1 -22144.337,E2 -22144.337} C_VEL
LIN {X 0,Y 185.975,Z 246.285,A -85,B 0,C 180,E1 -22148.695,E2 -22148.695} C_VEL
LIN {X 0,Y 185.708,Z 246.347,A -85,B 0,C 180,E1 -22153.195,E2 -22153.195} C_VEL
LIN {X 0,Y 186.381,Z 248.635,A -85,B 0,C 180,E1 -22153.98,E2 -22153.98} C_VEL
LIN {X 0,Y 188.348,Z 251.057,A -85,B 0,C 180,E1 -22155.696,E2 -22155.696} C_VEL
LIN {X 0,Y 190.553,Z 252.413,A -85,B 0,C 180,E1 -22157.328,E2 -22157.328} C_VEL
LIN {X 0,Y 192.098,Z 255.359,A -85,B 0,C 180,E1 -22158.562,E2 -22158.562} C_VEL
LIN {X 0,Y 194.508,Z 257.545,A -85,B 0,C 180,E1 -22160.156,E2 -22160.156} C_VEL
LIN {X 0,Y 195.172,Z 258.438,A -85,B 0,C 180,E1 -22160.595,E2 -22160.595} C_VEL
LIN {X 0,Y 197.538,Z 261.668,A -85,B 0,C 180,E1 -22162.087,E2 -22162.087} C_VEL
LIN {X 0,Y 199.096,Z 263.298,A -85,B 0,C 180,E1 -22162.974,E2 -22162.974} C_VEL
LIN {X 0,Y 201.789,Z 266.961,A -85,B 0,C 180,E1 -22164.48,E2 -22164.48} C_VEL
LIN {X 0,Y 203.592,Z 269.367,A -85,B 0,C 180,E1 -22165.431,E2 -22165.431} C_VEL
LIN {X 0,Y 206.622,Z 273.483,A -85,B 0,C 180,E1 -22166.946,E2 -22166.946} C_VEL
LIN {X 0,Y 211.634,Z 280.611,A -85,B 0,C 180,E1 -22169.261,E2 -22169.261} C_VEL
LIN {X 0,Y 217.975,Z 290.649,A -85,B 0,C 180,E1 -22171.937,E2 -22171.937} C_VEL
LIN {X 0,Y 224.556,Z 302.37,A -85,B 0,C 180,E1 -22174.454,E2 -22174.454} C_VEL
LIN {X 0,Y 226.005,Z 305.185,A -85,B 0,C 180,E1 -22174.983,E2 -22174.983} C_VEL
LIN {X 0,Y 223.224,Z 347.711,A -85,B 0,C 180,E1 -22176.276,E2 -22176.276} C_VEL
LIN {X 0,Y 221.639,Z 360.601,A -85,B 0,C 180,E1 -22176.993,E2 -22176.993} C_VEL
LIN {X 0,Y 219.204,Z 373.524,A -85,B 0,C 180,E1 -22178.05,E2 -22178.05} C_VEL
LIN {X 0,Y 216.137,Z 385.802,A -85,B 0,C 180,E1 -22179.446,E2 -22179.446} C_VEL
LIN {X 0,Y 212.794,Z 396.434,A -85,B 0,C 180,E1 -22181.034,E2 -22181.034} C_VEL
LIN {X 0,Y 208.963,Z 406.688,A -85,B 0,C 180,E1 -22182.99,E2 -22182.99} C_VEL
LIN {X 0,Y 204.81,Z 416.145,A -85,B 0,C 180,E1 -22185.299,E2 -22185.299} C_VEL
LIN {X 0,Y 200.312,Z 425.209,A -85,B 0,C 180,E1 -22188.197,E2 -22188.197} C_VEL
LIN {X 0,Y 196.338,Z 432.404,A -85,B 0,C 180,E1 -22191.217,E2 -22191.217} C_VEL
LIN {X 0,Y 192.869,Z 438.048,A -85,B 0,C 180,E1 -22194.339,E2 -22194.339} C_VEL
LIN {X 0,Y 189.969,Z 442.399,A -85,B 0,C 180,E1 -22197.562,E2 -22197.562} C_VEL
LIN {X 0,Y 187.565,Z 445.593,A -85,B 0,C 180,E1 -22200.852,E2 -22200.852} C_VEL
LIN {X 0,Y 186.278,Z 447.149,A -85,B 0,C 180,E1 -22203.083,E2 -22203.083} C_VEL
LIN {X 0,Y 185.105,Z 448.346,A -85,B 0,C 180,E1 -22205.677,E2 -22205.677} C_VEL
LIN {X 0,Y 183.73,Z 449.117,A -85,B 0,C 180,E1 -22209.866,E2 -22209.866} C_VEL
LIN {X 0,Y 183.18,Z 448.59,A -85,B 0,C 180,E1 -22213.573,E2 -22213.573} C_VEL
LIN {X 0,Y 182.983,Z 447.263,A -85,B 0,C 180,E1 -22216.679,E2 -22216.679} C_VEL
LIN {X 0,Y 183.047,Z 445.816,A -85,B 0,C 180,E1 -22218.935,E2 -22218.935} C_VEL
LIN {X 0,Y 183.497,Z 442.792,A -85,B 0,C 180,E1 -22222.299,E2 -22222.299} C_VEL
LIN {X 0,Y 184.248,Z 438.704,A -85,B 0,C 180,E1 -22225.627,E2 -22225.627} C_VEL
LIN {X 0,Y 185.465,Z 432.451,A -85,B 0,C 180,E1 -22229.46,E2 -22229.46} C_VEL
LIN {X 0,Y 186.961,Z 425.644,A -85,B 0,C 180,E1 -22232.696,E2 -22232.696} C_VEL
LIN {X 0,Y 188.954,Z 417.086,A -85,B 0,C 180,E1 -22235.873,E2 -22235.873} C_VEL
LIN {X 0,Y 190.979,Z 408.314,A -85,B 0,C 180,E1 -22238.467,E2 -22238.467} C_VEL
LIN {X 0,Y 193.329,Z 397.754,A -85,B 0,C 180,E1 -22240.947,E2 -22240.947} C_VEL
LIN {X 0,Y 195.507,Z 386.561,A -85,B 0,C 180,E1 -22242.986,E2 -22242.986} C_VEL
LIN {X 0,Y 197.076,Z 376.357,A -85,B 0,C 180,E1 -22244.458,E2 -22244.458} C_VEL
LIN {X 0,Y 198.413,Z 365.515,A -85,B 0,C 180,E1 -22245.672,E2 -22245.672} C_VEL
LIN {X 0,Y 199.711,Z 352.624,A -85,B 0,C 180,E1 -22246.693,E2 -22246.693} C_VEL
LIN {X 0,Y 200.564,Z 338.977,A -85,B 0,C 180,E1 -22247.341,E2 -22247.341} C_VEL
LIN {X 0,Y 202.839,Z 282.527,A -85,B 0,C 180,E1 -22249.246,E2 -22249.246} C_VEL
LIN {X 0,Y 196.006,Z 266.763,A -85,B 0,C 180,E1 -22250.963,E2 -22250.963} C_VEL
LIN {X 0,Y 187.079,Z 249.862,A -85,B 0,C 180,E1 -22253.276,E2 -22253.276} C_VEL
LIN {X 0,Y 185.761,Z 247.064,A -85,B 0,C 180,E1 -22253.654,E2 -22253.654} C_VEL
LIN {X 0,Y 185.65,Z 246.357,A -85,B 0,C 180,E1 -22253.732,E2 -22253.732} C_VEL
LIN {X 0,Y 185.55,Z 246.37,A -85,B 0,C 180,E1 -22259.501,E2 -22259.501} C_VEL
LIN {X 0,Y 185.503,Z 246.375,A -85,B 0,C 180,E1 -22264.634,E2 -22264.634} C_VEL
LIN {X 0,Y 185.506,Z 246.37,A -85,B 0,C 180,E1 -22267.316,E2 -22267.316} C_VEL
LIN {X 0,Y 185.468,Z 246.379,A -85,B 0,C 180,E1 -22270.722,E2 -22270.722} C_VEL
LIN {X 0,Y 185.462,Z 246.381,A -85,B 0,C 180,E1 -22276.057,E2 -22276.057} C_VEL
LIN {X 0,Y 185.462,Z 246.368,A -85,B 0,C 180,E1 -22279.893,E2 -22279.893} C_VEL
LIN {X 0,Y 185.507,Z 246.359,A -85,B 0,C 180,E1 -22282.715,E2 -22282.715} C_VEL
LIN {X 0,Y 185.546,Z 246.367,A -85,B 0,C 180,E1 -22287.974,E2 -22287.974} C_VEL
LIN {X 0,Y 185.648,Z 246.328,A -85,B 0,C 180,E1 -22291.732,E2 -22291.732} C_VEL
LIN {X 0,Y 192.607,Z 274.144,A -85,B 0,C 180,E1 -22293.873,E2 -22293.873} C_VEL
LIN {X 0,Y 189.082,Z 348.137,A -85,B 0,C 180,E1 -22298.924,E2 -22298.924} C_VEL
LIN {X 0,Y 188.281,Z 362.625,A -85,B 0,C 180,E1 -22300.369,E2 -22300.369} C_VEL
LIN {X 0,Y 187.308,Z 376.461,A -85,B 0,C 180,E1 -22302.25,E2 -22302.25} C_VEL
LIN {X 0,Y 186.312,Z 388.872,A -85,B 0,C 180,E1 -22304.408,E2 -22304.408} C_VEL
LIN {X 0,Y 185.517,Z 400.205,A -85,B 0,C 180,E1 -22306.861,E2 -22306.861} C_VEL
LIN {X 0,Y 184.76,Z 410.47,A -85,B 0,C 180,E1 -22309.59,E2 -22309.59} C_VEL
LIN {X 0,Y 184.224,Z 420.029,A -85,B 0,C 180,E1 -22312.709,E2 -22312.709} C_VEL
LIN {X 0,Y 183.844,Z 428.588,A -85,B 0,C 180,E1 -22316.164,E2 -22316.164} C_VEL
LIN {X 0,Y 183.731,Z 434.134,A -85,B 0,C 180,E1 -22318.904,E2 -22318.904} C_VEL
LIN {X 0,Y 183.794,Z 439.604,A -85,B 0,C 180,E1 -22322.191,E2 -22322.191} C_VEL
LIN {X 0,Y 184.379,Z 443.999,A -85,B 0,C 180,E1 -22325.468,E2 -22325.468} C_VEL
LIN {X 0,Y 185.355,Z 447.423,A -85,B 0,C 180,E1 -22328.723,E2 -22328.723} C_VEL
LIN {X 0,Y 187.347,Z 450.644,A -85,B 0,C 180,E1 -22333.007,E2 -22333.007} C_VEL
LIN {X 0,Y 189.132,Z 451.73,A -85,B 0,C 180,E1 -22335.076,E2 -22335.076} C_VEL
LIN {X 0,Y 193.181,Z 452.778,A -85,B 0,C 180,E1 -22339.112,E2 -22339.112} C_VEL
LIN {X 0,Y 198.349,Z 452.412,A -85,B 0,C 180,E1 -22342.939,E2 -22342.939} C_VEL
LIN {X 0,Y 204.531,Z 450.655,A -85,B 0,C 180,E1 -22346.532,E2 -22346.532} C_VEL
LIN {X 0,Y 211.67,Z 447.41,A -85,B 0,C 180,E1 -22349.87,E2 -22349.87} C_VEL
LIN {X 0,Y 219.73,Z 442.595,A -85,B 0,C 180,E1 -22352.938,E2 -22352.938} C_VEL
LIN {X 0,Y 226.272,Z 437.877,A -85,B 0,C 180,E1 -22355.072,E2 -22355.072} C_VEL
LIN {X 0,Y 234.485,Z 431.014,A -85,B 0,C 180,E1 -22357.368,E2 -22357.368} C_VEL
LIN {X 0,Y 243.147,Z 422.446,A -85,B 0,C 180,E1 -22359.486,E2 -22359.486} C_VEL
LIN {X 0,Y 248.636,Z 416.318,A -85,B 0,C 180,E1 -22360.676,E2 -22360.676} C_VEL
LIN {X 0,Y 249.493,Z 415.256,A -85,B 0,C 180,E1 -22361.091,E2 -22361.091} C_VEL
LIN {X 0,Y 249.663,Z 414.993,A -85,B 0,C 180,E1 -22361.827,E2 -22361.827} C_VEL
LIN {X 0,Y 248.811,Z 415.967,A -85,B 0,C 180,E1 -22362.832,E2 -22362.832} C_VEL
LIN {X 0,Y 247.573,Z 417.423,A -85,B 0,C 180,E1 -22363.573,E2 -22363.573} C_VEL
LIN {X 0,Y 244.522,Z 421.028,A -85,B 0,C 180,E1 -22364.836,E2 -22364.836} C_VEL
LIN {X 0,Y 240.269,Z 425.812,A -85,B 0,C 180,E1 -22366.107,E2 -22366.107} C_VEL
LIN {X 0,Y 238.149,Z 427.996,A -85,B 0,C 180,E1 -22366.558,E2 -22366.558} C_VEL
LIN {X 0,Y 228.416,Z 437.222,A -85,B 0,C 180,E1 -22368.582,E2 -22368.582} C_VEL
LIN {X 0,Y 220.862,Z 443.513,A -85,B 0,C 180,E1 -22370.473,E2 -22370.473} C_VEL
LIN {X 0,Y 213.768,Z 448.769,A -85,B 0,C 180,E1 -22372.537,E2 -22372.537} C_VEL
LIN {X 0,Y 205.066,Z 454.396,A -85,B 0,C 180,E1 -22375.562,E2 -22375.562} C_VEL
LIN {X 0,Y 199.173,Z 457.592,A -85,B 0,C 180,E1 -22378.04,E2 -22378.04} C_VEL
LIN {X 0,Y 192.21,Z 460.683,A -85,B 0,C 180,E1 -22381.616,E2 -22381.616} C_VEL
LIN {X 0,Y 186.659,Z 462.43,A -85,B 0,C 180,E1 -22385.531,E2 -22385.531} C_VEL
LIN {X 0,Y 182.211,Z 462.876,A -85,B 0,C 180,E1 -22389.685,E2 -22389.685} C_VEL
LIN {X 0,Y 179.153,Z 462.038,A -85,B 0,C 180,E1 -22394.059,E2 -22394.059} C_VEL
LIN {X 0,Y 177.522,Z 459.909,A -85,B 0,C 180,E1 -22398.581,E2 -22398.581} C_VEL
LIN {X 0,Y 177.147,Z 457.181,A -85,B 0,C 180,E1 -22402.303,E2 -22402.303} C_VEL
LIN {X 0,Y 176.522,Z 460.314,A -85,B 0,C 180,E1 -22405.43,E2 -22405.43} C_VEL
LIN {X 0,Y 176.421,Z 462.039,A -85,B 0,C 180,E1 -22407.714,E2 -22407.714} C_VEL
LIN {X 0,Y 176.502,Z 463.336,A -85,B 0,C 180,E1 -22409.997,E2 -22409.997} C_VEL
LIN {X 0,Y 176.145,Z 464.588,A -85,B 0,C 180,E1 -22414.078,E2 -22414.078} C_VEL
LIN {X 0,Y 176.148,Z 464.697,A -85,B 0,C 180,E1 -22416.872,E2 -22416.872} C_VEL
LIN {X 0,Y 176.927,Z 463.613,A -85,B 0,C 180,E1 -22421.453,E2 -22421.453} C_VEL
LIN {X 0,Y 177.643,Z 462.484,A -85,B 0,C 180,E1 -22423.729,E2 -22423.729} C_VEL
LIN {X 0,Y 178.632,Z 460.915,A -85,B 0,C 180,E1 -22425.983,E2 -22425.983} C_VEL
LIN {X 0,Y 180.827,Z 457.797,A -85,B 0,C 180,E1 -22429.288,E2 -22429.288} C_VEL
LIN {X 0,Y 184.287,Z 452.453,A -85,B 0,C 180,E1 -22433.286,E2 -22433.286} C_VEL
LIN {X 0,Y 187.896,Z 446.285,A -85,B 0,C 180,E1 -22436.667,E2 -22436.667} C_VEL
LIN {X 0,Y 192.044,Z 439.126,A -85,B 0,C 180,E1 -22439.604,E2 -22439.604} C_VEL
LIN {X 0,Y 196.711,Z 430.267,A -85,B 0,C 180,E1 -22442.403,E2 -22442.403} C_VEL
LIN {X 0,Y 200.988,Z 421.154,A -85,B 0,C 180,E1 -22444.623,E2 -22444.623} C_VEL
LIN {X 0,Y 205.015,Z 411.04,A -85,B 0,C 180,E1 -22446.554,E2 -22446.554} C_VEL
LIN {X 0,Y 209.002,Z 399.836,A -85,B 0,C 180,E1 -22448.159,E2 -22448.159} C_VEL
LIN {X 0,Y 212.434,Z 388.185,A -85,B 0,C 180,E1 -22449.401,E2 -22449.401} C_VEL
LIN {X 0,Y 215.194,Z 375.416,A -85,B 0,C 180,E1 -22450.394,E2 -22450.394} C_VEL
LIN {X 0,Y 217.142,Z 362.008,A -85,B 0,C 180,E1 -22451.101,E2 -22451.101} C_VEL
LIN {X 0,Y 219.857,Z 320.389,A -85,B 0,C 180,E1 -22452.421,E2 -22452.421} C_VEL
LIN {X 0,Y 218.465,Z 304.279,A -85,B 0,C 180,E1 -22453.629,E2 -22453.629} C_VEL
LIN {X 0,Y 217.432,Z 301.315,A -85,B 0,C 180,E1 -22454.096,E2 -22454.096} C_VEL
LIN {X 0,Y 211.823,Z 291.555,A -85,B 0,C 180,E1 -22456.468,E2 -22456.468} C_VEL
LIN {X 0,Y 205.408,Z 281.669,A -85,B 0,C 180,E1 -22459.452,E2 -22459.452} C_VEL
LIN {X 0,Y 201.458,Z 276.232,A -85,B 0,C 180,E1 -22461.467,E2 -22461.467} C_VEL
LIN {X 0,Y 199.217,Z 273.136,A -85,B 0,C 180,E1 -22462.697,E2 -22462.697} C_VEL
LIN {X 0,Y 195.787,Z 268.543,A -85,B 0,C 180,E1 -22464.718,E2 -22464.718} C_VEL
LIN {X 0,Y 193.182,Z 265.331,A -85,B 0,C 180,E1 -22466.384,E2 -22466.384} C_VEL
LIN {X 0,Y 192.27,Z 263.973,A -85,B 0,C 180,E1 -22467.021,E2 -22467.021} C_VEL
LIN {X 0,Y 189.662,Z 261.308,A -85,B 0,C 180,E1 -22468.867,E2 -22468.867} C_VEL
LIN {X 0,Y 188.289,Z 258.841,A -85,B 0,C 180,E1 -22470.013,E2 -22470.013} C_VEL
LIN {X 0,Y 185.623,Z 256.776,A -85,B 0,C 180,E1 -22472.175,E2 -22472.175} C_VEL
LIN {X 0,Y 183.931,Z 254.034,A -85,B 0,C 180,E1 -22473.858,E2 -22473.858} C_VEL
LIN {X 0,Y 183.652,Z 253.21,A -85,B 0,C 180,E1 -22474.196,E2 -22474.196} C_VEL
LIN {X 0,Y 180.596,Z 251.424,A -85,B 0,C 180,E1 -22477.401,E2 -22477.401} C_VEL
LIN {X 0,Y 178.987,Z 249.15,A -85,B 0,C 180,E1 -22479.658,E2 -22479.658} C_VEL
LIN {X 0,Y 178.541,Z 247.221,A -85,B 0,C 180,E1 -22480.706,E2 -22480.706} C_VEL
LIN {X 0,Y 178.63,Z 247.186,A -85,B 0,C 180,E1 -22486.346,E2 -22486.346} C_VEL
LIN {X 0,Y 178.896,Z 247.196,A -85,B 0,C 180,E1 -22490.959,E2 -22490.959} C_VEL
LIN {X 0,Y 179.119,Z 247.158,A -85,B 0,C 180,E1 -22497.752,E2 -22497.752} C_VEL
LIN {X 0,Y 179.338,Z 247.122,A -85,B 0,C 180,E1 -22500.001,E2 -22500.001} C_VEL
LIN {X 0,Y 178.893,Z 247.277,A -85,B 0,C 180,E1 -22506.273,E2 -22506.273} C_VEL
LIN {X 0,Y 179.535,Z 249.407,A -85,B 0,C 180,E1 -22507.451,E2 -22507.451} C_VEL
LIN {X 0,Y 181.757,Z 252.031,A -85,B 0,C 180,E1 -22510.288,E2 -22510.288} C_VEL
LIN {X 0,Y 183.867,Z 253.338,A -85,B 0,C 180,E1 -22512.416,E2 -22512.416} C_VEL
LIN {X 0,Y 185.235,Z 256.129,A -85,B 0,C 180,E1 -22513.858,E2 -22513.858} C_VEL
LIN {X 0,Y 187.481,Z 258.299,A -85,B 0,C 180,E1 -22515.771,E2 -22515.771} C_VEL
LIN {X 0,Y 188.542,Z 259.039,A -85,B 0,C 180,E1 -22516.583,E2 -22516.583} C_VEL
LIN {X 0,Y 190.476,Z 262.247,A -85,B 0,C 180,E1 -22518.139,E2 -22518.139} C_VEL
LIN {X 0,Y 192.856,Z 264.543,A -85,B 0,C 180,E1 -22519.769,E2 -22519.769} C_VEL
LIN {X 0,Y 195.241,Z 267.907,A -85,B 0,C 180,E1 -22521.358,E2 -22521.358} C_VEL
LIN {X 0,Y 196.68,Z 269.569,A -85,B 0,C 180,E1 -22522.223,E2 -22522.223} C_VEL
LIN {X 0,Y 200.847,Z 275.223,A -85,B 0,C 180,E1 -22524.603,E2 -22524.603} C_VEL
LIN {X 0,Y 205.983,Z 282.397,A -85,B 0,C 180,E1 -22527.229,E2 -22527.229} C_VEL
LIN {X 0,Y 212.767,Z 292.993,A -85,B 0,C 180,E1 -22530.342,E2 -22530.342} C_VEL
LIN {X 0,Y 218.856,Z 303.797,A -85,B 0,C 180,E1 -22532.869,E2 -22532.869} C_VEL
LIN {X 0,Y 220.977,Z 307.882,A -85,B 0,C 180,E1 -22533.698,E2 -22533.698} C_VEL
LIN {X 0,Y 218.309,Z 347.895,A -85,B 0,C 180,E1 -22534.944,E2 -22534.944} C_VEL
LIN {X 0,Y 216.74,Z 360.525,A -85,B 0,C 180,E1 -22535.652,E2 -22535.652} C_VEL
LIN {X 0,Y 214.389,Z 372.659,A -85,B 0,C 180,E1 -22536.628,E2 -22536.628} C_VEL
LIN {X 0,Y 211.487,Z 384.147,A -85,B 0,C 180,E1 -22537.889,E2 -22537.889} C_VEL
LIN {X 0,Y 207.872,Z 395.628,A -85,B 0,C 180,E1 -22539.565,E2 -22539.565} C_VEL
LIN {X 0,Y 203.537,Z 406.827,A -85,B 0,C 180,E1 -22541.698,E2 -22541.698} C_VEL
LIN {X 0,Y 199.62,Z 415.473,A -85,B 0,C 180,E1 -22543.805,E2 -22543.805} C_VEL
LIN {X 0,Y 195.693,Z 423.218,A -85,B 0,C 180,E1 -22546.2,E2 -22546.2} C_VEL
LIN {X 0,Y 191.235,Z 430.957,A -85,B 0,C 180,E1 -22549.286,E2 -22549.286} C_VEL
LIN {X 0,Y 187.714,Z 436.638,A -85,B 0,C 180,E1 -22552.257,E2 -22552.257} C_VEL
LIN {X 0,Y 184.72,Z 440.985,A -85,B 0,C 180,E1 -22555.204,E2 -22555.204} C_VEL
LIN {X 0,Y 182.342,Z 444.127,A -85,B 0,C 180,E1 -22557.99,E2 -22557.99} C_VEL
LIN {X 0,Y 179.677,Z 447.254,A -85,B 0,C 180,E1 -22562.009,E2 -22562.009} C_VEL
LIN {X 0,Y 178.182,Z 448.692,A -85,B 0,C 180,E1 -22565.121,E2 -22565.121} C_VEL
LIN {X 0,Y 176.817,Z 449.417,A -85,B 0,C 180,E1 -22569.042,E2 -22569.042} C_VEL
LIN {X 0,Y 176.105,Z 448.895,A -85,B 0,C 180,E1 -22573.297,E2 -22573.297} C_VEL
LIN {X 0,Y 175.911,Z 447.751,A -85,B 0,C 180,E1 -22576.133,E2 -22576.133} C_VEL
LIN {X 0,Y 175.915,Z 446.372,A -85,B 0,C 180,E1 -22578.48,E2 -22578.48} C_VEL
LIN {X 0,Y 176.347,Z 443.445,A -85,B 0,C 180,E1 -22581.984,E2 -22581.984} C_VEL
LIN {X 0,Y 177.117,Z 439.472,A -85,B 0,C 180,E1 -22585.451,E2 -22585.451} C_VEL
LIN {X 0,Y 178.338,Z 433.349,A -85,B 0,C 180,E1 -22589.438,E2 -22589.438} C_VEL
LIN {X 0,Y 179.831,Z 426.672,A -85,B 0,C 180,E1 -22592.803,E2 -22592.803} C_VEL
LIN {X 0,Y 181.854,Z 418.342,A -85,B 0,C 180,E1 -22596.103,E2 -22596.103} C_VEL
LIN {X 0,Y 183.958,Z 409.745,A -85,B 0,C 180,E1 -22598.793,E2 -22598.793} C_VEL
LIN {X 0,Y 186.363,Z 399.56,A -85,B 0,C 180,E1 -22601.331,E2 -22601.331} C_VEL
LIN {X 0,Y 188.579,Z 388.667,A -85,B 0,C 180,E1 -22603.472,E2 -22603.472} C_VEL
LIN {X 0,Y 190.531,Z 376.979,A -85,B 0,C 180,E1 -22605.239,E2 -22605.239} C_VEL
LIN {X 0,Y 191.902,Z 366.235,A -85,B 0,C 180,E1 -22606.491,E2 -22606.491} C_VEL
LIN {X 0,Y 193.255,Z 353.541,A -85,B 0,C 180,E1 -22607.542,E2 -22607.542} C_VEL
LIN {X 0,Y 194.197,Z 339.504,A -85,B 0,C 180,E1 -22608.236,E2 -22608.236} C_VEL
LIN {X 0,Y 196.548,Z 284.404,A -85,B 0,C 180,E1 -22610.142,E2 -22610.142} C_VEL
LIN {X 0,Y 190.24,Z 269.847,A -85,B 0,C 180,E1 -22611.818,E2 -22611.818} C_VEL
LIN {X 0,Y 181.94,Z 254.076,A -85,B 0,C 180,E1 -22614.084,E2 -22614.084} C_VEL
LIN {X 0,Y 180.017,Z 250.777,A -85,B 0,C 180,E1 -22614.629,E2 -22614.629} C_VEL
LIN {X 0,Y 178.641,Z 247.97,A -85,B 0,C 180,E1 -22615.05,E2 -22615.05} C_VEL
LIN {X 0,Y 178.507,Z 247.249,A -85,B 0,C 180,E1 -22615.16,E2 -22615.16} C_VEL
LIN {X 0,Y 178.466,Z 247.245,A -85,B 0,C 180,E1 -22620.796,E2 -22620.796} C_VEL
LIN {X 0,Y 178.489,Z 247.25,A -85,B 0,C 180,E1 -22624.219,E2 -22624.219} C_VEL
LIN {X 0,Y 178.393,Z 247.263,A -85,B 0,C 180,E1 -22629.078,E2 -22629.078} C_VEL
LIN {X 0,Y 178.399,Z 247.248,A -85,B 0,C 180,E1 -22632.048,E2 -22632.048} C_VEL
LIN {X 0,Y 178.397,Z 247.256,A -85,B 0,C 180,E1 -22635.166,E2 -22635.166} C_VEL
LIN {X 0,Y 178.403,Z 247.257,A -85,B 0,C 180,E1 -22638.463,E2 -22638.463} C_VEL
LIN {X 0,Y 178.425,Z 247.248,A -85,B 0,C 180,E1 -22643.783,E2 -22643.783} C_VEL
LIN {X 0,Y 178.491,Z 247.249,A -85,B 0,C 180,E1 -22646.547,E2 -22646.547} C_VEL
LIN {X 0,Y 178.605,Z 247.229,A -85,B 0,C 180,E1 -22651.606,E2 -22651.606} C_VEL
LIN {X 0,Y 185.472,Z 275.236,A -85,B 0,C 180,E1 -22653.782,E2 -22653.782} C_VEL
LIN {X 0,Y 181.981,Z 348.614,A -85,B 0,C 180,E1 -22659.057,E2 -22659.057} C_VEL
LIN {X 0,Y 181.15,Z 363.314,A -85,B 0,C 180,E1 -22660.597,E2 -22660.597} C_VEL
LIN {X 0,Y 180.114,Z 377.847,A -85,B 0,C 180,E1 -22662.69,E2 -22662.69} C_VEL
LIN {X 0,Y 179.113,Z 391.327,A -85,B 0,C 180,E1 -22665.223,E2 -22665.223} C_VEL
LIN {X 0,Y 178.257,Z 402.2,A -85,B 0,C 180,E1 -22667.765,E2 -22667.765} C_VEL
LIN {X 0,Y 177.511,Z 412.947,A -85,B 0,C 180,E1 -22670.887,E2 -22670.887} C_VEL
LIN {X 0,Y 177.04,Z 422.566,A -85,B 0,C 180,E1 -22674.316,E2 -22674.316} C_VEL
LIN {X 0,Y 176.825,Z 430.226,A -85,B 0,C 180,E1 -22677.722,E2 -22677.722} C_VEL
LIN {X 0,Y 176.738,Z 436.469,A -85,B 0,C 180,E1 -22681.139,E2 -22681.139} C_VEL
LIN {X 0,Y 177.136,Z 441.547,A -85,B 0,C 180,E1 -22684.551,E2 -22684.551} C_VEL
LIN {X 0,Y 178.382,Z 446.741,A -85,B 0,C 180,E1 -22689.067,E2 -22689.067} C_VEL
LIN {X 0,Y 180.456,Z 450.359,A -85,B 0,C 180,E1 -22693.513,E2 -22693.513} C_VEL
LIN {X 0,Y 184.248,Z 452.543,A -85,B 0,C 180,E1 -22697.767,E2 -22697.767} C_VEL
LIN {X 0,Y 189.094,Z 453.337,A -85,B 0,C 180,E1 -22701.818,E2 -22701.818} C_VEL
LIN {X 0,Y 194.942,Z 452.766,A -85,B 0,C 180,E1 -22705.634,E2 -22705.634} C_VEL
LIN {X 0,Y 201.914,Z 450.744,A -85,B 0,C 180,E1 -22709.163,E2 -22709.163} C_VEL
LIN {X 0,Y 209.786,Z 447.287,A -85,B 0,C 180,E1 -22712.412,E2 -22712.412} C_VEL
LIN {X 0,Y 218.515,Z 442.285,A -85,B 0,C 180,E1 -22715.375,E2 -22715.375} C_VEL
LIN {X 0,Y 225.558,Z 437.415,A -85,B 0,C 180,E1 -22717.415,E2 -22717.415} C_VEL
LIN {X 0,Y 234.333,Z 430.281,A -85,B 0,C 180,E1 -22719.592,E2 -22719.592} C_VEL
LIN {X 0,Y 243.531,Z 421.547,A -85,B 0,C 180,E1 -22721.586,E2 -22721.586} C_VEL
LIN {X 0,Y 251.603,Z 412.542,A -85,B 0,C 180,E1 -22723.116,E2 -22723.116} C_VEL
LIN {X 0,Y 254.619,Z 408.827,A -85,B 0,C 180,E1 -22723.634,E2 -22723.634} C_VEL
LIN {X 0,Y 253.822,Z 409.926,A -85,B 0,C 180,E1 -22723.951,E2 -22723.951} C_VEL
LIN {X 0,Y 244.99,Z 420.659,A -85,B 0,C 180,E1 -22725.343,E2 -22725.343} C_VEL
LIN {X 0,Y 238.149,Z 427.996,A -85,B 0,C 180,E1 -22726.558,E2 -22726.558} C_VEL
LIN {X 0,Y 234.179,Z 431.805,A -85,B 0,C 180,E1 -22727.133,E2 -22727.133} C_VEL
LIN {X 0,Y 226.773,Z 437.894,A -85,B 0,C 180,E1 -22727.801,E2 -22727.801} C_VEL
LIN {X 0,Y 219.246,Z 443.258,A -85,B 0,C 180,E1 -22728.616,E2 -22728.616} C_VEL
LIN {X 0,Y 215.146,Z 446.012,A -85,B 0,C 180,E1 -22729.427,E2 -22729.427} C_VEL
LIN {X 0,Y 205.938,Z 451.871,A -85,B 0,C 180,E1 -22732.098,E2 -22732.098} C_VEL
LIN {X 0,Y 197.215,Z 456.474,A -85,B 0,C 180,E1 -22735.235,E2 -22735.235} C_VEL
LIN {X 0,Y 189.457,Z 459.721,A -85,B 0,C 180,E1 -22738.71,E2 -22738.71} C_VEL
LIN {X 0,Y 182.942,Z 461.663,A -85,B 0,C 180,E1 -22742.546,E2 -22742.546} C_VEL
LIN {X 0,Y 177.719,Z 462.353,A -85,B 0,C 180,E1 -22746.703,E2 -22746.703} C_VEL
LIN {X 0,Y 173.729,Z 461.768,A -85,B 0,C 180,E1 -22751.115,E2 -22751.115} C_VEL
LIN {X 0,Y 171.352,Z 459.927,A -85,B 0,C 180,E1 -22755.751,E2 -22755.751} C_VEL
LIN {X 0,Y 170.359,Z 456.755,A -85,B 0,C 180,E1 -22760.499,E2 -22760.499} C_VEL
LIN {X 0,Y 170.264,Z 456.09,A -85,B 0,C 180,E1 -22761.541,E2 -22761.541} C_VEL
LIN {X 0,Y 169.451,Z 459.793,A -85,B 0,C 180,E1 -22765.239,E2 -22765.239} C_VEL
LIN {X 0,Y 169.345,Z 461.585,A -85,B 0,C 180,E1 -22767.619,E2 -22767.619} C_VEL
LIN {X 0,Y 169.433,Z 462.913,A -85,B 0,C 180,E1 -22769.997,E2 -22769.997} C_VEL
LIN {X 0,Y 169.068,Z 464.169,A -85,B 0,C 180,E1 -22773.925,E2 -22773.925} C_VEL
LIN {X 0,Y 169.094,Z 464.397,A -85,B 0,C 180,E1 -22777.16,E2 -22777.16} C_VEL
LIN {X 0,Y 169.953,Z 463.375,A -85,B 0,C 180,E1 -22781.93,E2 -22781.93} C_VEL
LIN {X 0,Y 170.706,Z 462.291,A -85,B 0,C 180,E1 -22784.299,E2 -22784.299} C_VEL
LIN {X 0,Y 171.798,Z 460.774,A -85,B 0,C 180,E1 -22786.637,E2 -22786.637} C_VEL
LIN {X 0,Y 174.123,Z 457.727,A -85,B 0,C 180,E1 -22790.062,E2 -22790.062} C_VEL
LIN {X 0,Y 177.644,Z 452.635,A -85,B 0,C 180,E1 -22794.077,E2 -22794.077} C_VEL
LIN {X 0,Y 181.574,Z 446.403,A -85,B 0,C 180,E1 -22797.673,E2 -22797.673} C_VEL
LIN {X 0,Y 185.9,Z 439.359,A -85,B 0,C 180,E1 -22800.686,E2 -22800.686} C_VEL
LIN {X 0,Y 190.778,Z 430.61,A -85,B 0,C 180,E1 -22803.541,E2 -22803.541} C_VEL
LIN {X 0,Y 195.209,Z 421.651,A -85,B 0,C 180,E1 -22805.803,E2 -22805.803} C_VEL
LIN {X 0,Y 199.386,Z 411.768,A -85,B 0,C 180,E1 -22807.763,E2 -22807.763} C_VEL
LIN {X 0,Y 203.51,Z 400.793,A -85,B 0,C 180,E1 -22809.384,E2 -22809.384} C_VEL
LIN {X 0,Y 207.314,Z 388.524,A -85,B 0,C 180,E1 -22810.733,E2 -22810.733} C_VEL
LIN {X 0,Y 210.171,Z 376.053,A -85,B 0,C 180,E1 -22811.729,E2 -22811.729} C_VEL
LIN {X 0,Y 212.163,Z 363.323,A -85,B 0,C 180,E1 -22812.428,E2 -22812.428} C_VEL
LIN {X 0,Y 213.704,Z 343.647,A -85,B 0,C 180,E1 -22813.095,E2 -22813.095} C_VEL
LIN {X 0,Y 215.121,Z 321.263,A -85,B 0,C 180,E1 -22813.798,E2 -22813.798} C_VEL
LIN {X 0,Y 213.913,Z 306.845,A -85,B 0,C 180,E1 -22814.932,E2 -22814.932} C_VEL
LIN {X 0,Y 209.913,Z 299.363,A -85,B 0,C 180,E1 -22816.709,E2 -22816.709} C_VEL
LIN {X 0,Y 204.558,Z 290.596,A -85,B 0,C 180,E1 -22819.249,E2 -22819.249} C_VEL
LIN {X 0,Y 199.407,Z 282.986,A -85,B 0,C 180,E1 -22821.941,E2 -22821.941} C_VEL
LIN {X 0,Y 196.212,Z 278.629,A -85,B 0,C 180,E1 -22823.769,E2 -22823.769} C_VEL
LIN {X 0,Y 193.364,Z 274.717,A -85,B 0,C 180,E1 -22825.543,E2 -22825.543} C_VEL
LIN {X 0,Y 190.532,Z 270.814,A -85,B 0,C 180,E1 -22827.498,E2 -22827.498} C_VEL
LIN {X 0,Y 187.435,Z 267.301,A -85,B 0,C 180,E1 -22829.814,E2 -22829.814} C_VEL
LIN {X 0,Y 186.246,Z 265.359,A -85,B 0,C 180,E1 -22830.841,E2 -22830.841} C_VEL
LIN {X 0,Y 183.441,Z 262.709,A -85,B 0,C 180,E1 -22833.304,E2 -22833.304} C_VEL
LIN {X 0,Y 182.009,Z 260.063,A -85,B 0,C 180,E1 -22834.866,E2 -22834.866} C_VEL
LIN {X 0,Y 179,Z 257.906,A -85,B 0,C 180,E1 -22838.251,E2 -22838.251} C_VEL
LIN {X 0,Y 177.482,Z 255.411,A -85,B 0,C 180,E1 -22840.619,E2 -22840.619} C_VEL
LIN {X 0,Y 177.056,Z 254.163,A -85,B 0,C 180,E1 -22841.486,E2 -22841.486} C_VEL
LIN {X 0,Y 173.607,Z 251.958,A -85,B 0,C 180,E1 -22851.855,E2 -22851.855} C_VEL
LIN {X 0,Y 174.361,Z 252.347,A -85,B 0,C 180,E1 -22858.846,E2 -22858.846} C_VEL
LIN {X 0,Y 177.51,Z 254.259,A -85,B 0,C 180,E1 -22865.61,E2 -22865.61} C_VEL
LIN {X 0,Y 178.6,Z 256.829,A -85,B 0,C 180,E1 -22867.49,E2 -22867.49} C_VEL
LIN {X 0,Y 180.927,Z 259.268,A -85,B 0,C 180,E1 -22870.414,E2 -22870.414} C_VEL
LIN {X 0,Y 182.223,Z 260.19,A -85,B 0,C 180,E1 -22871.753,E2 -22871.753} C_VEL
LIN {X 0,Y 183.995,Z 263.251,A -85,B 0,C 180,E1 -22873.619,E2 -22873.619} C_VEL
LIN {X 0,Y 186.679,Z 265.731,A -85,B 0,C 180,E1 -22875.91,E2 -22875.91} C_VEL
LIN {X 0,Y 188.989,Z 269.201,A -85,B 0,C 180,E1 -22877.797,E2 -22877.797} C_VEL
LIN {X 0,Y 190.838,Z 271.184,A -85,B 0,C 180,E1 -22879.121,E2 -22879.121} C_VEL
LIN {X 0,Y 193.775,Z 274.98,A -85,B 0,C 180,E1 -22881.109,E2 -22881.109} C_VEL
LIN {X 0,Y 198.5,Z 281.658,A -85,B 0,C 180,E1 -22883.958,E2 -22883.958} C_VEL
LIN {X 0,Y 202.956,Z 287.987,A -85,B 0,C 180,E1 -22886.339,E2 -22886.339} C_VEL
LIN {X 0,Y 209.349,Z 298.224,A -85,B 0,C 180,E1 -22889.427,E2 -22889.427} C_VEL
LIN {X 0,Y 215.355,Z 309.202,A -85,B 0,C 180,E1 -22892.057,E2 -22892.057} C_VEL
LIN {X 0,Y 216.196,Z 310.875,A -85,B 0,C 180,E1 -22892.409,E2 -22892.409} C_VEL
LIN {X 0,Y 213.543,Z 348.004,A -85,B 0,C 180,E1 -22893.555,E2 -22893.555} C_VEL
LIN {X 0,Y 211.906,Z 360.697,A -85,B 0,C 180,E1 -22894.263,E2 -22894.263} C_VEL
LIN {X 0,Y 209.335,Z 373.48,A -85,B 0,C 180,E1 -22895.306,E2 -22895.306} C_VEL
LIN {X 0,Y 206.501,Z 384.167,A -85,B 0,C 180,E1 -22896.486,E2 -22896.486} C_VEL
LIN {X 0,Y 203.084,Z 394.78,A -85,B 0,C 180,E1 -22898.018,E2 -22898.018} C_VEL
LIN {X 0,Y 199.165,Z 404.802,A -85,B 0,C 180,E1 -22899.874,E2 -22899.874} C_VEL
LIN {X 0,Y 194.532,Z 414.735,A -85,B 0,C 180,E1 -22902.22,E2 -22902.22} C_VEL
LIN {X 0,Y 190.335,Z 422.808,A -85,B 0,C 180,E1 -22904.697,E2 -22904.697} C_VEL
LIN {X 0,Y 185.66,Z 430.616,A -85,B 0,C 180,E1 -22907.789,E2 -22907.789} C_VEL
LIN {X 0,Y 182.382,Z 435.741,A -85,B 0,C 180,E1 -22910.417,E2 -22910.417} C_VEL
LIN {X 0,Y 178.648,Z 440.886,A -85,B 0,C 180,E1 -22913.839,E2 -22913.839} C_VEL
LIN {X 0,Y 175.758,Z 444.503,A -85,B 0,C 180,E1 -22917.112,E2 -22917.112} C_VEL
LIN {X 0,Y 173.153,Z 447.362,A -85,B 0,C 180,E1 -22920.856,E2 -22920.856} C_VEL
LIN {X 0,Y 171.316,Z 449.027,A -85,B 0,C 180,E1 -22924.493,E2 -22924.493} C_VEL
LIN {X 0,Y 169.941,Z 449.718,A -85,B 0,C 180,E1 -22928.152,E2 -22928.152} C_VEL
LIN {X 0,Y 169.379,Z 449.652,A -85,B 0,C 180,E1 -22930.616,E2 -22930.616} C_VEL
LIN {X 0,Y 169.05,Z 449.172,A -85,B 0,C 180,E1 -22933.084,E2 -22933.084} C_VEL
LIN {X 0,Y 168.839,Z 448.239,A -85,B 0,C 180,E1 -22935.54,E2 -22935.54} C_VEL
LIN {X 0,Y 168.793,Z 446.908,A -85,B 0,C 180,E1 -22937.987,E2 -22937.987} C_VEL
LIN {X 0,Y 169.18,Z 444.078,A -85,B 0,C 180,E1 -22941.643,E2 -22941.643} C_VEL
LIN {X 0,Y 169.95,Z 440.207,A -85,B 0,C 180,E1 -22945.258,E2 -22945.258} C_VEL
LIN {X 0,Y 170.947,Z 435.216,A -85,B 0,C 180,E1 -22948.825,E2 -22948.825} C_VEL
LIN {X 0,Y 172.37,Z 428.925,A -85,B 0,C 180,E1 -22952.339,E2 -22952.339} C_VEL
LIN {X 0,Y 174.377,Z 421.024,A -85,B 0,C 180,E1 -22955.785,E2 -22955.785} C_VEL
LIN {X 0,Y 176.467,Z 412.959,A -85,B 0,C 180,E1 -22958.592,E2 -22958.592} C_VEL
LIN {X 0,Y 178.872,Z 403.139,A -85,B 0,C 180,E1 -22961.332,E2 -22961.332} C_VEL
LIN {X 0,Y 181.38,Z 392.036,A -85,B 0,C 180,E1 -22963.731,E2 -22963.731} C_VEL
LIN {X 0,Y 183.471,Z 381.217,A -85,B 0,C 180,E1 -22965.556,E2 -22965.556} C_VEL
LIN {X 0,Y 185.091,Z 369.414,A -85,B 0,C 180,E1 -22967.116,E2 -22967.116} C_VEL
LIN {X 0,Y 186.679,Z 356.571,A -85,B 0,C 180,E1 -22968.281,E2 -22968.281} C_VEL
LIN {X 0,Y 187.675,Z 343.525,A -85,B 0,C 180,E1 -22969.055,E2 -22969.055} C_VEL
LIN {X 0,Y 190.274,Z 286.171,A -85,B 0,C 180,E1 -22971.107,E2 -22971.107} C_VEL
LIN {X 0,Y 184.368,Z 272.597,A -85,B 0,C 180,E1 -22972.764,E2 -22972.764} C_VEL
LIN {X 0,Y 175.615,Z 255.896,A -85,B 0,C 180,E1 -22975.317,E2 -22975.317} C_VEL
LIN {X 0,Y 172.739,Z 251.424,A -85,B 0,C 180,E1 -22976.178,E2 -22976.178} C_VEL
LIN {X 0,Y 171.521,Z 248.801,A -85,B 0,C 180,E1 -22976.591,E2 -22976.591} C_VEL
LIN {X 0,Y 171.408,Z 248.128,A -85,B 0,C 180,E1 -22976.7,E2 -22976.7} C_VEL
LIN {X 0,Y 171.423,Z 248.122,A -85,B 0,C 180,E1 -22980.574,E2 -22980.574} C_VEL
LIN {X 0,Y 171.398,Z 248.128,A -85,B 0,C 180,E1 -22985.036,E2 -22985.036} C_VEL
LIN {X 0,Y 171.349,Z 248.14,A -85,B 0,C 180,E1 -22988.802,E2 -22988.802} C_VEL
LIN {X 0,Y 171.325,Z 248.131,A -85,B 0,C 180,E1 -22994.219,E2 -22994.219} C_VEL
LIN {X 0,Y 171.336,Z 248.131,A -85,B 0,C 180,E1 -22998.981,E2 -22998.981} C_VEL
LIN {X 0,Y 171.366,Z 248.114,A -85,B 0,C 180,E1 -23002.034,E2 -23002.034} C_VEL
LIN {X 0,Y 171.404,Z 248.129,A -85,B 0,C 180,E1 -23005.094,E2 -23005.094} C_VEL
LIN {X 0,Y 171.543,Z 248.084,A -85,B 0,C 180,E1 -23011.211,E2 -23011.211} C_VEL
LIN {X 0,Y 171.586,Z 248.251,A -85,B 0,C 180,E1 -23011.453,E2 -23011.453} C_VEL
LIN {X 0,Y 175.971,Z 266.11,A -85,B 0,C 180,E1 -23012.906,E2 -23012.906} C_VEL
LIN {X 0,Y 178.382,Z 275.687,A -85,B 0,C 180,E1 -23013.667,E2 -23013.667} C_VEL
LIN {X 0,Y 174.907,Z 347.795,A -85,B 0,C 180,E1 -23019.107,E2 -23019.107} C_VEL
LIN {X 0,Y 174.096,Z 362.543,A -85,B 0,C 180,E1 -23020.699,E2 -23020.699} C_VEL
LIN {X 0,Y 173.181,Z 375.548,A -85,B 0,C 180,E1 -23022.584,E2 -23022.584} C_VEL
LIN {X 0,Y 172.227,Z 388.141,A -85,B 0,C 180,E1 -23024.921,E2 -23024.921} C_VEL
LIN {X 0,Y 171.414,Z 399.554,A -85,B 0,C 180,E1 -23027.569,E2 -23027.569} C_VEL
LIN {X 0,Y 170.728,Z 409.96,A -85,B 0,C 180,E1 -23030.522,E2 -23030.522} C_VEL
LIN {X 0,Y 170.177,Z 419.948,A -85,B 0,C 180,E1 -23034.032,E2 -23034.032} C_VEL
LIN {X 0,Y 169.893,Z 428.23,A -85,B 0,C 180,E1 -23037.629,E2 -23037.629} C_VEL
LIN {X 0,Y 169.808,Z 434.865,A -85,B 0,C 180,E1 -23041.185,E2 -23041.185} C_VEL
LIN {X 0,Y 170.173,Z 440.267,A -85,B 0,C 180,E1 -23044.737,E2 -23044.737} C_VEL
LIN {X 0,Y 171.036,Z 444.633,A -85,B 0,C 180,E1 -23048.268,E2 -23048.268} C_VEL
LIN {X 0,Y 172.3,Z 448.069,A -85,B 0,C 180,E1 -23051.767,E2 -23051.767} C_VEL
LIN {X 0,Y 173.576,Z 449.891,A -85,B 0,C 180,E1 -23054.059,E2 -23054.059} C_VEL
LIN {X 0,Y 177.509,Z 452.526,A -85,B 0,C 180,E1 -23058.465,E2 -23058.465} C_VEL
LIN {X 0,Y 182.547,Z 453.783,A -85,B 0,C 180,E1 -23062.643,E2 -23062.643} C_VEL
LIN {X 0,Y 188.622,Z 453.644,A -85,B 0,C 180,E1 -23066.558,E2 -23066.558} C_VEL
LIN {X 0,Y 195.87,Z 452.129,A -85,B 0,C 180,E1 -23070.154,E2 -23070.154} C_VEL
LIN {X 0,Y 204.012,Z 449.241,A -85,B 0,C 180,E1 -23073.448,E2 -23073.448} C_VEL
LIN {X 0,Y 213.031,Z 444.834,A -85,B 0,C 180,E1 -23076.429,E2 -23076.429} C_VEL
LIN {X 0,Y 222.805,Z 438.789,A -85,B 0,C 180,E1 -23079.114,E2 -23079.114} C_VEL
LIN {X 0,Y 231.993,Z 431.963,A -85,B 0,C 180,E1 -23081.215,E2 -23081.215} C_VEL
LIN {X 0,Y 240.295,Z 424.707,A -85,B 0,C 180,E1 -23082.901,E2 -23082.901} C_VEL
LIN {X 0,Y 241.83,Z 423.249,A -85,B 0,C 180,E1 -23083.188,E2 -23083.188} C_VEL
LIN {X 0,Y 243.231,Z 421.957,A -85,B 0,C 180,E1 -23083.748,E2 -23083.748} C_VEL
LIN {X 0,Y 234.421,Z 430.607,A -85,B 0,C 180,E1 -23085.206,E2 -23085.206} C_VEL
LIN {X 0,Y 224.669,Z 438.942,A -85,B 0,C 180,E1 -23087.125,E2 -23087.125} C_VEL
LIN {X 0,Y 215.146,Z 446.012,A -85,B 0,C 180,E1 -23089.427,E2 -23089.427} C_VEL
LIN {X 0,Y 210.954,Z 448.648,A -85,B 0,C 180,E1 -23090.32,E2 -23090.32} C_VEL
LIN {X 0,Y 202.996,Z 452.657,A -85,B 0,C 180,E1 -23091.543,E2 -23091.543} C_VEL
LIN {X 0,Y 195.137,Z 455.917,A -85,B 0,C 180,E1 -23092.957,E2 -23092.957} C_VEL
LIN {X 0,Y 191.169,Z 457.387,A -85,B 0,C 180,E1 -23094.154,E2 -23094.154} C_VEL
LIN {X 0,Y 183.432,Z 460.002,A -85,B 0,C 180,E1 -23097.559,E2 -23097.559} C_VEL
LIN {X 0,Y 176.668,Z 461.47,A -85,B 0,C 180,E1 -23101.483,E2 -23101.483} C_VEL
LIN {X 0,Y 171.246,Z 461.724,A -85,B 0,C 180,E1 -23105.767,E2 -23105.767} C_VEL
LIN {X 0,Y 167.079,Z 460.745,A -85,B 0,C 180,E1 -23110.333,E2 -23110.333} C_VEL
LIN {X 0,Y 164.598,Z 458.565,A -85,B 0,C 180,E1 -23115.153,E2 -23115.153} C_VEL
LIN {X 0,Y 163.567,Z 455.054,A -85,B 0,C 180,E1 -23120.101,E2 -23120.101} C_VEL
LIN {X 0,Y 163.49,Z 454.797,A -85,B 0,C 180,E1 -23120.565,E2 -23120.565} C_VEL
LIN {X 0,Y 162.383,Z 459.272,A -85,B 0,C 180,E1 -23125.031,E2 -23125.031} C_VEL
LIN {X 0,Y 162.271,Z 461.121,A -85,B 0,C 180,E1 -23127.515,E2 -23127.515} C_VEL
LIN {X 0,Y 162.365,Z 462.491,A -85,B 0,C 180,E1 -23129.997,E2 -23129.997} C_VEL
LIN {X 0,Y 162.008,Z 463.766,A -85,B 0,C 180,E1 -23133.846,E2 -23133.846} C_VEL
LIN {X 0,Y 162.02,Z 464.094,A -85,B 0,C 180,E1 -23137.474,E2 -23137.474} C_VEL
LIN {X 0,Y 162.962,Z 463.139,A -85,B 0,C 180,E1 -23142.45,E2 -23142.45} C_VEL
LIN {X 0,Y 163.791,Z 462.088,A -85,B 0,C 180,E1 -23144.916,E2 -23144.916} C_VEL
LIN {X 0,Y 164.995,Z 460.638,A -85,B 0,C 180,E1 -23147.345,E2 -23147.345} C_VEL
LIN {X 0,Y 167.44,Z 457.656,A -85,B 0,C 180,E1 -23150.899,E2 -23150.899} C_VEL
LIN {X 0,Y 170.464,Z 453.649,A -85,B 0,C 180,E1 -23154.345,E2 -23154.345} C_VEL
LIN {X 0,Y 174.625,Z 447.501,A -85,B 0,C 180,E1 -23158.219,E2 -23158.219} C_VEL
LIN {X 0,Y 179.054,Z 440.822,A -85,B 0,C 180,E1 -23161.334,E2 -23161.334} C_VEL
LIN {X 0,Y 184.021,Z 432.556,A -85,B 0,C 180,E1 -23164.283,E2 -23164.283} C_VEL
LIN {X 0,Y 188.586,Z 424.046,A -85,B 0,C 180,E1 -23166.6,E2 -23166.6} C_VEL
LIN {X 0,Y 193.361,Z 413.6,A -85,B 0,C 180,E1 -23168.824,E2 -23168.824} C_VEL
LIN {X 0,Y 197.573,Z 403.236,A -85,B 0,C 180,E1 -23170.477,E2 -23170.477} C_VEL
LIN {X 0,Y 201.42,Z 391.761,A -85,B 0,C 180,E1 -23171.857,E2 -23171.857} C_VEL
LIN {X 0,Y 204.828,Z 378.681,A -85,B 0,C 180,E1 -23172.993,E2 -23172.993} C_VEL
LIN {X 0,Y 207.104,Z 366.096,A -85,B 0,C 180,E1 -23173.761,E2 -23173.761} C_VEL
LIN {X 0,Y 208.535,Z 351.539,A -85,B 0,C 180,E1 -23174.322,E2 -23174.322} C_VEL
LIN {X 0,Y 210.512,Z 322.346,A -85,B 0,C 180,E1 -23175.235,E2 -23175.235} C_VEL
LIN {X 0,Y 209.612,Z 310.271,A -85,B 0,C 180,E1 -23176.206,E2 -23176.206} C_VEL
LIN {X 0,Y 204.024,Z 300.182,A -85,B 0,C 180,E1 -23178.878,E2 -23178.878} C_VEL
LIN {X 0,Y 198.409,Z 291.393,A -85,B 0,C 180,E1 -23181.831,E2 -23181.831} C_VEL
LIN {X 0,Y 193.817,Z 284.78,A -85,B 0,C 180,E1 -23184.537,E2 -23184.537} C_VEL
LIN {X 0,Y 190.759,Z 280.539,A -85,B 0,C 180,E1 -23186.555,E2 -23186.555} C_VEL
LIN {X 0,Y 187.93,Z 276.609,A -85,B 0,C 180,E1 -23188.635,E2 -23188.635} C_VEL
LIN {X 0,Y 185.165,Z 273.105,A -85,B 0,C 180,E1 -23190.872,E2 -23190.872} C_VEL
LIN {X 0,Y 184.379,Z 271.917,A -85,B 0,C 180,E1 -23191.579,E2 -23191.579} C_VEL
LIN {X 0,Y 181.518,Z 268.885,A -85,B 0,C 180,E1 -23194.265,E2 -23194.265} C_VEL
LIN {X 0,Y 180.352,Z 266.756,A -85,B 0,C 180,E1 -23195.608,E2 -23195.608} C_VEL
LIN {X 0,Y 177.58,Z 264.563,A -85,B 0,C 180,E1 -23198.925,E2 -23198.925} C_VEL
LIN {X 0,Y 176.06,Z 261.777,A -85,B 0,C 180,E1 -23201.528,E2 -23201.528} C_VEL
LIN {X 0,Y 175.872,Z 261.11,A -85,B 0,C 180,E1 -23201.959,E2 -23201.959} C_VEL
LIN {X 0,Y 172.725,Z 259.01,A -85,B 0,C 180,E1 -23211.813,E2 -23211.813} C_VEL
LIN {X 0,Y 173.661,Z 259.482,A -85,B 0,C 180,E1 -23219.421,E2 -23219.421} C_VEL
LIN {X 0,Y 176.251,Z 261.283,A -85,B 0,C 180,E1 -23225.083,E2 -23225.083} C_VEL
LIN {X 0,Y 177.617,Z 264.087,A -85,B 0,C 180,E1 -23227.443,E2 -23227.443} C_VEL
LIN {X 0,Y 180.053,Z 266.411,A -85,B 0,C 180,E1 -23230.465,E2 -23230.465} C_VEL
LIN {X 0,Y 180.68,Z 267.029,A -85,B 0,C 180,E1 -23231.15,E2 -23231.15} C_VEL
LIN {X 0,Y 182.726,Z 270.307,A -85,B 0,C 180,E1 -23233.343,E2 -23233.343} C_VEL
LIN {X 0,Y 184.9,Z 272.434,A -85,B 0,C 180,E1 -23235.272,E2 -23235.272} C_VEL
LIN {X 0,Y 187.323,Z 275.916,A -85,B 0,C 180,E1 -23237.309,E2 -23237.309} C_VEL
LIN {X 0,Y 188.853,Z 277.734,A -85,B 0,C 180,E1 -23238.459,E2 -23238.459} C_VEL
LIN {X 0,Y 192.207,Z 282.314,A -85,B 0,C 180,E1 -23240.816,E2 -23240.816} C_VEL
LIN {X 0,Y 195.851,Z 287.547,A -85,B 0,C 180,E1 -23243.101,E2 -23243.101} C_VEL
LIN {X 0,Y 200.199,Z 293.91,A -85,B 0,C 180,E1 -23245.54,E2 -23245.54} C_VEL
LIN {X 0,Y 206.285,Z 304.023,A -85,B 0,C 180,E1 -23248.627,E2 -23248.627} C_VEL
LIN {X 0,Y 211.45,Z 313.683,A -85,B 0,C 180,E1 -23251.011,E2 -23251.011} C_VEL
LIN {X 0,Y 208.881,Z 348.695,A -85,B 0,C 180,E1 -23252.124,E2 -23252.124} C_VEL
LIN {X 0,Y 207.032,Z 361.865,A -85,B 0,C 180,E1 -23252.874,E2 -23252.874} C_VEL
LIN {X 0,Y 204.539,Z 373.708,A -85,B 0,C 180,E1 -23253.854,E2 -23253.854} C_VEL
LIN {X 0,Y 201.148,Z 385.98,A -85,B 0,C 180,E1 -23255.247,E2 -23255.247} C_VEL
LIN {X 0,Y 196.979,Z 397.838,A -85,B 0,C 180,E1 -23257.078,E2 -23257.078} C_VEL
LIN {X 0,Y 192.524,Z 408.187,A -85,B 0,C 180,E1 -23259.133,E2 -23259.133} C_VEL
LIN {X 0,Y 187.831,Z 417.517,A -85,B 0,C 180,E1 -23261.558,E2 -23261.558} C_VEL
LIN {X 0,Y 182.637,Z 426.504,A -85,B 0,C 180,E1 -23264.615,E2 -23264.615} C_VEL
LIN {X 0,Y 178.011,Z 433.611,A -85,B 0,C 180,E1 -23267.846,E2 -23267.846} C_VEL
LIN {X 0,Y 173.924,Z 439.202,A -85,B 0,C 180,E1 -23271.224,E2 -23271.224} C_VEL
LIN {X 0,Y 170.454,Z 443.505,A -85,B 0,C 180,E1 -23274.747,E2 -23274.747} C_VEL
LIN {X 0,Y 168.431,Z 445.749,A -85,B 0,C 180,E1 -23277.153,E2 -23277.153} C_VEL
LIN {X 0,Y 166.699,Z 447.472,A -85,B 0,C 180,E1 -23279.611,E2 -23279.611} C_VEL
LIN {X 0,Y 164.452,Z 449.37,A -85,B 0,C 180,E1 -23283.827,E2 -23283.827} C_VEL
LIN {X 0,Y 163.112,Z 450.019,A -85,B 0,C 180,E1 -23287.186,E2 -23287.186} C_VEL
LIN {X 0,Y 162.455,Z 450,A -85,B 0,C 180,E1 -23289.755,E2 -23289.755} C_VEL
LIN {X 0,Y 161.974,Z 449.501,A -85,B 0,C 180,E1 -23292.667,E2 -23292.667} C_VEL
LIN {X 0,Y 161.681,Z 447.441,A -85,B 0,C 180,E1 -23297.45,E2 -23297.45} C_VEL
LIN {X 0,Y 162.023,Z 444.708,A -85,B 0,C 180,E1 -23301.271,E2 -23301.271} C_VEL
LIN {X 0,Y 162.793,Z 440.936,A -85,B 0,C 180,E1 -23305.05,E2 -23305.05} C_VEL
LIN {X 0,Y 163.792,Z 436.053,A -85,B 0,C 180,E1 -23308.773,E2 -23308.773} C_VEL
LIN {X 0,Y 165.243,Z 429.902,A -85,B 0,C 180,E1 -23312.44,E2 -23312.44} C_VEL
LIN {X 0,Y 167.291,Z 422.186,A -85,B 0,C 180,E1 -23316.031,E2 -23316.031} C_VEL
LIN {X 0,Y 169.427,Z 414.285,A -85,B 0,C 180,E1 -23318.952,E2 -23318.952} C_VEL
LIN {X 0,Y 172.152,Z 403.694,A -85,B 0,C 180,E1 -23322.057,E2 -23322.057} C_VEL
LIN {X 0,Y 174.786,Z 392.554,A -85,B 0,C 180,E1 -23324.557,E2 -23324.557} C_VEL
LIN {X 0,Y 176.954,Z 381.781,A -85,B 0,C 180,E1 -23326.441,E2 -23326.441} C_VEL
LIN {X 0,Y 178.656,Z 370.054,A -85,B 0,C 180,E1 -23328.049,E2 -23328.049} C_VEL
LIN {X 0,Y 180.335,Z 357.038,A -85,B 0,C 180,E1 -23329.273,E2 -23329.273} C_VEL
LIN {X 0,Y 181.446,Z 343.212,A -85,B 0,C 180,E1 -23330.106,E2 -23330.106} C_VEL
LIN {X 0,Y 184.085,Z 287.991,A -85,B 0,C 180,E1 -23332.123,E2 -23332.123} C_VEL
LIN {X 0,Y 178.581,Z 275.46,A -85,B 0,C 180,E1 -23333.759,E2 -23333.759} C_VEL
LIN {X 0,Y 170.544,Z 260.141,A -85,B 0,C 180,E1 -23336.244,E2 -23336.244} C_VEL
LIN {X 0,Y 165.987,Z 252.771,A -85,B 0,C 180,E1 -23337.723,E2 -23337.723} C_VEL
LIN {X 0,Y 164.523,Z 250.014,A -85,B 0,C 180,E1 -23338.242,E2 -23338.242} C_VEL
LIN {X 0,Y 164.337,Z 249.016,A -85,B 0,C 180,E1 -23338.413,E2 -23338.413} C_VEL
LIN {X 0,Y 164.363,Z 249.001,A -85,B 0,C 180,E1 -23341.219,E2 -23341.219} C_VEL
LIN {X 0,Y 164.286,Z 249.01,A -85,B 0,C 180,E1 -23346.795,E2 -23346.795} C_VEL
LIN {X 0,Y 164.292,Z 249.019,A -85,B 0,C 180,E1 -23349.919,E2 -23349.919} C_VEL
LIN {X 0,Y 164.286,Z 249.002,A -85,B 0,C 180,E1 -23353.343,E2 -23353.343} C_VEL
LIN {X 0,Y 164.267,Z 249.021,A -85,B 0,C 180,E1 -23356.799,E2 -23356.799} C_VEL
LIN {X 0,Y 164.295,Z 248.996,A -85,B 0,C 180,E1 -23360.356,E2 -23360.356} C_VEL
LIN {X 0,Y 164.332,Z 249.012,A -85,B 0,C 180,E1 -23366.221,E2 -23366.221} C_VEL
LIN {X 0,Y 164.503,Z 248.959,A -85,B 0,C 180,E1 -23371.26,E2 -23371.26} C_VEL
LIN {X 0,Y 168.727,Z 266.578,A -85,B 0,C 180,E1 -23372.783,E2 -23372.783} C_VEL
LIN {X 0,Y 171.231,Z 276.55,A -85,B 0,C 180,E1 -23373.601,E2 -23373.601} C_VEL
LIN {X 0,Y 167.805,Z 348.164,A -85,B 0,C 180,E1 -23379.305,E2 -23379.305} C_VEL
LIN {X 0,Y 167.01,Z 362.757,A -85,B 0,C 180,E1 -23380.965,E2 -23380.965} C_VEL
LIN {X 0,Y 166.041,Z 376.546,A -85,B 0,C 180,E1 -23383.082,E2 -23383.082} C_VEL
LIN {X 0,Y 165.129,Z 388.98,A -85,B 0,C 180,E1 -23385.519,E2 -23385.519} C_VEL
LIN {X 0,Y 164.302,Z 400.166,A -85,B 0,C 180,E1 -23388.276,E2 -23388.276} C_VEL
LIN {X 0,Y 163.68,Z 410.258,A -85,B 0,C 180,E1 -23391.292,E2 -23391.292} C_VEL
LIN {X 0,Y 163.232,Z 419.134,A -85,B 0,C 180,E1 -23394.518,E2 -23394.518} C_VEL
LIN {X 0,Y 162.986,Z 427.321,A -85,B 0,C 180,E1 -23398.146,E2 -23398.146} C_VEL
LIN {X 0,Y 162.928,Z 434.096,A -85,B 0,C 180,E1 -23401.853,E2 -23401.853} C_VEL
LIN {X 0,Y 163.505,Z 440.495,A -85,B 0,C 180,E1 -23406.168,E2 -23406.168} C_VEL
LIN {X 0,Y 164.733,Z 445.557,A -85,B 0,C 180,E1 -23410.513,E2 -23410.513} C_VEL
LIN {X 0,Y 166.73,Z 449.282,A -85,B 0,C 180,E1 -23414.649,E2 -23414.649} C_VEL
LIN {X 0,Y 170.791,Z 452.366,A -85,B 0,C 180,E1 -23419.22,E2 -23419.22} C_VEL
LIN {X 0,Y 176.038,Z 454.037,A -85,B 0,C 180,E1 -23423.53,E2 -23423.53} C_VEL
LIN {X 0,Y 182.345,Z 454.377,A -85,B 0,C 180,E1 -23427.549,E2 -23427.549} C_VEL
LIN {X 0,Y 189.847,Z 453.379,A -85,B 0,C 180,E1 -23431.216,E2 -23431.216} C_VEL
LIN {X 0,Y 198.283,Z 451.042,A -85,B 0,C 180,E1 -23434.549,E2 -23434.549} C_VEL
LIN {X 0,Y 207.593,Z 447.22,A -85,B 0,C 180,E1 -23437.545,E2 -23437.545} C_VEL
LIN {X 0,Y 217.655,Z 441.87,A -85,B 0,C 180,E1 -23440.225,E2 -23440.225} C_VEL
LIN {X 0,Y 225.7,Z 436.692,A -85,B 0,C 180,E1 -23442.027,E2 -23442.027} C_VEL
LIN {X 0,Y 231.073,Z 432.807,A -85,B 0,C 180,E1 -23443.115,E2 -23443.115} C_VEL
LIN {X 0,Y 232.571,Z 431.636,A -85,B 0,C 180,E1 -23443.508,E2 -23443.508} C_VEL
LIN {X 0,Y 222.461,Z 439.653,A -85,B 0,C 180,E1 -23445.335,E2 -23445.335} C_VEL
LIN {X 0,Y 212.986,Z 446.133,A -85,B 0,C 180,E1 -23447.431,E2 -23447.431} C_VEL
LIN {X 0,Y 202.864,Z 451.986,A -85,B 0,C 180,E1 -23450.138,E2 -23450.138} C_VEL
LIN {X 0,Y 195.857,Z 455.433,A -85,B 0,C 180,E1 -23452.407,E2 -23452.407} C_VEL
LIN {X 0,Y 191.169,Z 457.387,A -85,B 0,C 180,E1 -23454.154,E2 -23454.154} C_VEL
LIN {X 0,Y 187.248,Z 458.698,A -85,B 0,C 180,E1 -23455.447,E2 -23455.447} C_VEL
LIN {X 0,Y 179.653,Z 460.305,A -85,B 0,C 180,E1 -23457.385,E2 -23457.385} C_VEL
LIN {X 0,Y 173.778,Z 460.955,A -85,B 0,C 180,E1 -23459.075,E2 -23459.075} C_VEL
LIN {X 0,Y 170.195,Z 461.161,A -85,B 0,C 180,E1 -23460.617,E2 -23460.617} C_VEL
LIN {X 0,Y 169.28,Z 461.161,A -85,B 0,C 180,E1 -23461.199,E2 -23461.199} C_VEL
LIN {X 0,Y 164.842,Z 460.959,A -85,B 0,C 180,E1 -23464.761,E2 -23464.761} C_VEL
LIN {X 0,Y 160.5,Z 459.576,A -85,B 0,C 180,E1 -23469.491,E2 -23469.491} C_VEL
LIN {X 0,Y 157.897,Z 457.022,A -85,B 0,C 180,E1 -23474.508,E2 -23474.508} C_VEL
LIN {X 0,Y 156.787,Z 453.435,A -85,B 0,C 180,E1 -23479.505,E2 -23479.505} C_VEL
LIN {X 0,Y 155.429,Z 458.201,A -85,B 0,C 180,E1 -23484.133,E2 -23484.133} C_VEL
LIN {X 0,Y 155.18,Z 460.633,A -85,B 0,C 180,E1 -23487.401,E2 -23487.401} C_VEL
LIN {X 0,Y 155.295,Z 462.065,A -85,B 0,C 180,E1 -23489.997,E2 -23489.997} C_VEL
LIN {X 0,Y 154.95,Z 463.352,A -85,B 0,C 180,E1 -23493.768,E2 -23493.768} C_VEL
LIN {X 0,Y 154.961,Z 463.773,A -85,B 0,C 180,E1 -23497.817,E2 -23497.817} C_VEL
LIN {X 0,Y 155.369,Z 463.541,A -85,B 0,C 180,E1 -23500.421,E2 -23500.421} C_VEL
LIN {X 0,Y 156.899,Z 461.886,A -85,B 0,C 180,E1 -23505.587,E2 -23505.587} C_VEL
LIN {X 0,Y 158.224,Z 460.486,A -85,B 0,C 180,E1 -23508.112,E2 -23508.112} C_VEL
LIN {X 0,Y 160.783,Z 457.562,A -85,B 0,C 180,E1 -23511.808,E2 -23511.808} C_VEL
LIN {X 0,Y 163.993,Z 453.628,A -85,B 0,C 180,E1 -23515.373,E2 -23515.373} C_VEL
LIN {X 0,Y 167.7,Z 448.575,A -85,B 0,C 180,E1 -23518.809,E2 -23518.809} C_VEL
LIN {X 0,Y 172.204,Z 442.229,A -85,B 0,C 180,E1 -23522.04,E2 -23522.04} C_VEL
LIN {X 0,Y 177.355,Z 434.331,A -85,B 0,C 180,E1 -23525.067,E2 -23525.067} C_VEL
LIN {X 0,Y 182.006,Z 426.301,A -85,B 0,C 180,E1 -23527.454,E2 -23527.454} C_VEL
LIN {X 0,Y 186.96,Z 416.526,A -85,B 0,C 180,E1 -23529.717,E2 -23529.717} C_VEL
LIN {X 0,Y 191.121,Z 406.918,A -85,B 0,C 180,E1 -23531.442,E2 -23531.442} C_VEL
LIN {X 0,Y 195.641,Z 394.773,A -85,B 0,C 180,E1 -23533.039,E2 -23533.039} C_VEL
LIN {X 0,Y 199.128,Z 382.945,A -85,B 0,C 180,E1 -23534.188,E2 -23534.188} C_VEL
LIN {X 0,Y 201.764,Z 370.799,A -85,B 0,C 180,E1 -23535.035,E2 -23535.035} C_VEL
LIN {X 0,Y 203.635,Z 356.917,A -85,B 0,C 180,E1 -23535.672,E2 -23535.672} C_VEL
LIN {X 0,Y 206.056,Z 323.617,A -85,B 0,C 180,E1 -23536.725,E2 -23536.725} C_VEL
LIN {X 0,Y 205.392,Z 313.961,A -85,B 0,C 180,E1 -23537.528,E2 -23537.528} C_VEL
LIN {X 0,Y 200.618,Z 305.243,A -85,B 0,C 180,E1 -23539.956,E2 -23539.956} C_VEL
LIN {X 0,Y 195.664,Z 297.191,A -85,B 0,C 180,E1 -23542.717,E2 -23542.717} C_VEL
LIN {X 0,Y 191.272,Z 290.688,A -85,B 0,C 180,E1 -23545.447,E2 -23545.447} C_VEL
LIN {X 0,Y 188.531,Z 286.729,A -85,B 0,C 180,E1 -23547.371,E2 -23547.371} C_VEL
LIN {X 0,Y 185.784,Z 282.886,A -85,B 0,C 180,E1 -23549.492,E2 -23549.492} C_VEL
LIN {X 0,Y 183.05,Z 279.091,A -85,B 0,C 180,E1 -23551.862,E2 -23551.862} C_VEL
LIN {X 0,Y 179.534,Z 274.816,A -85,B 0,C 180,E1 -23555.384,E2 -23555.384} C_VEL
LIN {X 0,Y 178.673,Z 273.438,A -85,B 0,C 180,E1 -23556.418,E2 -23556.418} C_VEL
LIN {X 0,Y 175.939,Z 270.892,A -85,B 0,C 180,E1 -23560.01,E2 -23560.01} C_VEL
LIN {X 0,Y 174.687,Z 268.161,A -85,B 0,C 180,E1 -23562.438,E2 -23562.438} C_VEL
LIN {X 0,Y 171.845,Z 266.052,A -85,B 0,C 180,E1 -23571.771,E2 -23571.771} C_VEL
LIN {X 0,Y 172.782,Z 266.541,A -85,B 0,C 180,E1 -23579.418,E2 -23579.418} C_VEL
LIN {X 0,Y 174.994,Z 268.108,A -85,B 0,C 180,E1 -23584.463,E2 -23584.463} C_VEL
LIN {X 0,Y 176.625,Z 271.283,A -85,B 0,C 180,E1 -23587.359,E2 -23587.359} C_VEL
LIN {X 0,Y 179.144,Z 273.798,A -85,B 0,C 180,E1 -23590.519,E2 -23590.519} C_VEL
LIN {X 0,Y 181.511,Z 277.388,A -85,B 0,C 180,E1 -23593.114,E2 -23593.114} C_VEL
LIN {X 0,Y 183.071,Z 278.958,A -85,B 0,C 180,E1 -23594.548,E2 -23594.548} C_VEL
LIN {X 0,Y 185.69,Z 282.663,A -85,B 0,C 180,E1 -23596.827,E2 -23596.827} C_VEL
LIN {X 0,Y 187.215,Z 284.76,A -85,B 0,C 180,E1 -23598.033,E2 -23598.033} C_VEL
LIN {X 0,Y 189.919,Z 288.507,A -85,B 0,C 180,E1 -23600.009,E2 -23600.009} C_VEL
LIN {X 0,Y 194.901,Z 295.778,A -85,B 0,C 180,E1 -23603.22,E2 -23603.22} C_VEL
LIN {X 0,Y 201.181,Z 306.02,A -85,B 0,C 180,E1 -23606.73,E2 -23606.73} C_VEL
LIN {X 0,Y 206.909,Z 316.764,A -85,B 0,C 180,E1 -23609.591,E2 -23609.591} C_VEL
LIN {X 0,Y 204.42,Z 348.659,A -85,B 0,C 180,E1 -23610.594,E2 -23610.594} C_VEL
LIN {X 0,Y 202.632,Z 361.323,A -85,B 0,C 180,E1 -23611.299,E2 -23611.299} C_VEL
LIN {X 0,Y 200.023,Z 373.329,A -85,B 0,C 180,E1 -23612.263,E2 -23612.263} C_VEL
LIN {X 0,Y 196.945,Z 384.313,A -85,B 0,C 180,E1 -23613.478,E2 -23613.478} C_VEL
LIN {X 0,Y 193.17,Z 395.203,A -85,B 0,C 180,E1 -23615.059,E2 -23615.059} C_VEL
LIN {X 0,Y 188.797,Z 405.488,A -85,B 0,C 180,E1 -23616.99,E2 -23616.99} C_VEL
LIN {X 0,Y 183.921,Z 415.104,A -85,B 0,C 180,E1 -23619.308,E2 -23619.308} C_VEL
LIN {X 0,Y 179.317,Z 423.232,A -85,B 0,C 180,E1 -23621.873,E2 -23621.873} C_VEL
LIN {X 0,Y 174.982,Z 429.897,A -85,B 0,C 180,E1 -23624.532,E2 -23624.532} C_VEL
LIN {X 0,Y 171.151,Z 435.25,A -85,B 0,C 180,E1 -23627.249,E2 -23627.249} C_VEL
LIN {X 0,Y 166.86,Z 440.674,A -85,B 0,C 180,E1 -23630.822,E2 -23630.822} C_VEL
LIN {X 0,Y 162.709,Z 445.271,A -85,B 0,C 180,E1 -23635.155,E2 -23635.155} C_VEL
LIN {X 0,Y 160.327,Z 447.583,A -85,B 0,C 180,E1 -23638.266,E2 -23638.266} C_VEL
LIN {X 0,Y 157.617,Z 449.712,A -85,B 0,C 180,E1 -23643.1,E2 -23643.1} C_VEL
LIN {X 0,Y 156.353,Z 450.319,A -85,B 0,C 180,E1 -23646.14,E2 -23646.14} C_VEL
LIN {X 0,Y 155.567,Z 450.348,A -85,B 0,C 180,E1 -23648.816,E2 -23648.816} C_VEL
LIN {X 0,Y 154.941,Z 449.809,A -85,B 0,C 180,E1 -23652.28,E2 -23652.28} C_VEL
LIN {X 0,Y 154.584,Z 447.973,A -85,B 0,C 180,E1 -23656.864,E2 -23656.864} C_VEL
LIN {X 0,Y 154.866,Z 445.335,A -85,B 0,C 180,E1 -23660.864,E2 -23660.864} C_VEL
LIN {X 0,Y 155.615,Z 441.663,A -85,B 0,C 180,E1 -23664.821,E2 -23664.821} C_VEL
LIN {X 0,Y 156.642,Z 436.883,A -85,B 0,C 180,E1 -23668.717,E2 -23668.717} C_VEL
LIN {X 0,Y 158.126,Z 430.848,A -85,B 0,C 180,E1 -23672.55,E2 -23672.55} C_VEL
LIN {X 0,Y 160.217,Z 423.326,A -85,B 0,C 180,E1 -23676.299,E2 -23676.299} C_VEL
LIN {X 0,Y 162.895,Z 413.841,A -85,B 0,C 180,E1 -23679.94,E2 -23679.94} C_VEL
LIN {X 0,Y 165.539,Z 403.923,A -85,B 0,C 180,E1 -23682.927,E2 -23682.927} C_VEL
LIN {X 0,Y 168.23,Z 393.06,A -85,B 0,C 180,E1 -23685.448,E2 -23685.448} C_VEL
LIN {X 0,Y 170.489,Z 382.33,A -85,B 0,C 180,E1 -23687.392,E2 -23687.392} C_VEL
LIN {X 0,Y 172.273,Z 370.669,A -85,B 0,C 180,E1 -23689.051,E2 -23689.051} C_VEL
LIN {X 0,Y 174.016,Z 357.802,A -85,B 0,C 180,E1 -23690.311,E2 -23690.311} C_VEL
LIN {X 0,Y 175.189,Z 344.201,A -85,B 0,C 180,E1 -23691.167,E2 -23691.167} C_VEL
LIN {X 0,Y 177.833,Z 289.669,A -85,B 0,C 180,E1 -23693.24,E2 -23693.24} C_VEL
LIN {X 0,Y 173.132,Z 278.992,A -85,B 0,C 180,E1 -23694.726,E2 -23694.726} C_VEL
LIN {X 0,Y 165.736,Z 264.623,A -85,B 0,C 180,E1 -23697.158,E2 -23697.158} C_VEL
LIN {X 0,Y 159.651,Z 254.404,A -85,B 0,C 180,E1 -23699.295,E2 -23699.295} C_VEL
LIN {X 0,Y 157.795,Z 251.696,A -85,B 0,C 180,E1 -23699.968,E2 -23699.968} C_VEL
LIN {X 0,Y 157.32,Z 249.879,A -85,B 0,C 180,E1 -23700.279,E2 -23700.279} C_VEL
LIN {X 0,Y 157.265,Z 249.883,A -85,B 0,C 180,E1 -23706.446,E2 -23706.446} C_VEL
LIN {X 0,Y 157.196,Z 249.886,A -85,B 0,C 180,E1 -23712.119,E2 -23712.119} C_VEL
LIN {X 0,Y 157.196,Z 249.899,A -85,B 0,C 180,E1 -23717.883,E2 -23717.883} C_VEL
LIN {X 0,Y 157.265,Z 249.878,A -85,B 0,C 180,E1 -23723.557,E2 -23723.557} C_VEL
LIN {X 0,Y 157.299,Z 249.883,A -85,B 0,C 180,E1 -23728.098,E2 -23728.098} C_VEL
LIN {X 0,Y 157.47,Z 249.834,A -85,B 0,C 180,E1 -23731.132,E2 -23731.132} C_VEL
LIN {X 0,Y 161.335,Z 266.303,A -85,B 0,C 180,E1 -23732.616,E2 -23732.616} C_VEL
LIN {X 0,Y 164.109,Z 277.454,A -85,B 0,C 180,E1 -23733.566,E2 -23733.566} C_VEL
LIN {X 0,Y 160.686,Z 348.979,A -85,B 0,C 180,E1 -23739.602,E2 -23739.602} C_VEL
LIN {X 0,Y 159.923,Z 362.73,A -85,B 0,C 180,E1 -23741.254,E2 -23741.254} C_VEL
LIN {X 0,Y 159.04,Z 375.635,A -85,B 0,C 180,E1 -23743.307,E2 -23743.307} C_VEL
LIN {X 0,Y 158.036,Z 389.596,A -85,B 0,C 180,E1 -23746.17,E2 -23746.17} C_VEL
LIN {X 0,Y 157.261,Z 400.666,A -85,B 0,C 180,E1 -23749.05,E2 -23749.05} C_VEL
LIN {X 0,Y 156.656,Z 410.814,A -85,B 0,C 180,E1 -23752.265,E2 -23752.265} C_VEL
LIN {X 0,Y 156.277,Z 419.221,A -85,B 0,C 180,E1 -23755.486,E2 -23755.486} C_VEL
LIN {X 0,Y 156.103,Z 427.532,A -85,B 0,C 180,E1 -23759.354,E2 -23759.354} C_VEL
LIN {X 0,Y 156.188,Z 435.253,A -85,B 0,C 180,E1 -23763.87,E2 -23763.87} C_VEL
LIN {X 0,Y 156.895,Z 440.634,A -85,B 0,C 180,E1 -23767.722,E2 -23767.722} C_VEL
LIN {X 0,Y 158.565,Z 446.257,A -85,B 0,C 180,E1 -23772.803,E2 -23772.803} C_VEL
LIN {X 0,Y 159.919,Z 448.52,A -85,B 0,C 180,E1 -23775.288,E2 -23775.288} C_VEL
LIN {X 0,Y 164.13,Z 452.003,A -85,B 0,C 180,E1 -23780.032,E2 -23780.032} C_VEL
LIN {X 0,Y 169.561,Z 454.129,A -85,B 0,C 180,E1 -23784.486,E2 -23784.486} C_VEL
LIN {X 0,Y 176.127,Z 454.957,A -85,B 0,C 180,E1 -23788.609,E2 -23788.609} C_VEL
LIN {X 0,Y 183.89,Z 454.476,A -85,B 0,C 180,E1 -23792.347,E2 -23792.347} C_VEL
LIN {X 0,Y 188.085,Z 453.753,A -85,B 0,C 180,E1 -23794.089,E2 -23794.089} C_VEL
LIN {X 0,Y 197.306,Z 451.223,A -85,B 0,C 180,E1 -23797.267,E2 -23797.267} C_VEL
LIN {X 0,Y 207.272,Z 447.284,A -85,B 0,C 180,E1 -23800.108,E2 -23800.108} C_VEL
LIN {X 0,Y 215.252,Z 443.318,A -85,B 0,C 180,E1 -23802.015,E2 -23802.015} C_VEL
LIN {X 0,Y 220.445,Z 440.357,A -85,B 0,C 180,E1 -23803.106,E2 -23803.106} C_VEL
LIN {X 0,Y 219.903,Z 440.796,A -85,B 0,C 180,E1 -23803.634,E2 -23803.634} C_VEL
LIN {X 0,Y 210.629,Z 446.58,A -85,B 0,C 180,E1 -23805.514,E2 -23805.514} C_VEL
LIN {X 0,Y 200.044,Z 452.182,A -85,B 0,C 180,E1 -23808.122,E2 -23808.122} C_VEL
LIN {X 0,Y 190.316,Z 456.346,A -85,B 0,C 180,E1 -23811.111,E2 -23811.111} C_VEL
LIN {X 0,Y 181.519,Z 459.181,A -85,B 0,C 180,E1 -23814.493,E2 -23814.493} C_VEL
LIN {X 0,Y 173.799,Z 460.782,A -85,B 0,C 180,E1 -23818.283,E2 -23818.283} C_VEL
LIN {X 0,Y 169.28,Z 461.161,A -85,B 0,C 180,E1 -23821.199,E2 -23821.199} C_VEL
LIN {X 0,Y 166.294,Z 461.12,A -85,B 0,C 180,E1 -23822.936,E2 -23822.936} C_VEL
LIN {X 0,Y 160.212,Z 460.171,A -85,B 0,C 180,E1 -23825.66,E2 -23825.66} C_VEL
LIN {X 0,Y 154.707,Z 458.456,A -85,B 0,C 180,E1 -23828.592,E2 -23828.592} C_VEL
LIN {X 0,Y 152.709,Z 457.225,A -85,B 0,C 180,E1 -23830.616,E2 -23830.616} C_VEL
LIN {X 0,Y 151.24,Z 455.335,A -85,B 0,C 180,E1 -23833.808,E2 -23833.808} C_VEL
LIN {X 0,Y 150.175,Z 452.005,A -85,B 0,C 180,E1 -23838.354,E2 -23838.354} C_VEL
LIN {X 0,Y 148.516,Z 457.101,A -85,B 0,C 180,E1 -23843.204,E2 -23843.204} C_VEL
LIN {X 0,Y 148.093,Z 460.138,A -85,B 0,C 180,E1 -23847.277,E2 -23847.277} C_VEL
LIN {X 0,Y 148.225,Z 461.634,A -85,B 0,C 180,E1 -23849.997,E2 -23849.997} C_VEL
LIN {X 0,Y 147.881,Z 462.869,A -85,B 0,C 180,E1 -23853.611,E2 -23853.611} C_VEL
LIN {X 0,Y 147.926,Z 463.442,A -85,B 0,C 180,E1 -23858.191,E2 -23858.191} C_VEL
LIN {X 0,Y 148.353,Z 463.269,A -85,B 0,C 180,E1 -23860.92,E2 -23860.92} C_VEL
LIN {X 0,Y 150.036,Z 461.683,A -85,B 0,C 180,E1 -23866.32,E2 -23866.32} C_VEL
LIN {X 0,Y 151.459,Z 460.317,A -85,B 0,C 180,E1 -23868.951,E2 -23868.951} C_VEL
LIN {X 0,Y 154.178,Z 457.463,A -85,B 0,C 180,E1 -23872.793,E2 -23872.793} C_VEL
LIN {X 0,Y 157.579,Z 453.608,A -85,B 0,C 180,E1 -23876.484,E2 -23876.484} C_VEL
LIN {X 0,Y 161.499,Z 448.642,A -85,B 0,C 180,E1 -23880.026,E2 -23880.026} C_VEL
LIN {X 0,Y 166.243,Z 442.419,A -85,B 0,C 180,E1 -23883.335,E2 -23883.335} C_VEL
LIN {X 0,Y 171.59,Z 434.648,A -85,B 0,C 180,E1 -23886.43,E2 -23886.43} C_VEL
LIN {X 0,Y 176.447,Z 426.742,A -85,B 0,C 180,E1 -23888.85,E2 -23888.85} C_VEL
LIN {X 0,Y 182.078,Z 416.071,A -85,B 0,C 180,E1 -23891.373,E2 -23891.373} C_VEL
LIN {X 0,Y 187.036,Z 405.023,A -85,B 0,C 180,E1 -23893.291,E2 -23893.291} C_VEL
LIN {X 0,Y 191.139,Z 394.227,A -85,B 0,C 180,E1 -23894.681,E2 -23894.681} C_VEL
LIN {X 0,Y 194.757,Z 382.337,A -85,B 0,C 180,E1 -23895.821,E2 -23895.821} C_VEL
LIN {X 0,Y 197.555,Z 369.562,A -85,B 0,C 180,E1 -23896.69,E2 -23896.69} C_VEL
LIN {X 0,Y 199.344,Z 356.368,A -85,B 0,C 180,E1 -23897.29,E2 -23897.29} C_VEL
LIN {X 0,Y 201.747,Z 324.607,A -85,B 0,C 180,E1 -23898.297,E2 -23898.297} C_VEL
LIN {X 0,Y 201.293,Z 317.606,A -85,B 0,C 180,E1 -23898.905,E2 -23898.905} C_VEL
LIN {X 0,Y 196.677,Z 309.149,A -85,B 0,C 180,E1 -23901.423,E2 -23901.423} C_VEL
LIN {X 0,Y 191.88,Z 301.169,A -85,B 0,C 180,E1 -23904.32,E2 -23904.32} C_VEL
LIN {X 0,Y 186.769,Z 293.438,A -85,B 0,C 180,E1 -23907.888,E2 -23907.888} C_VEL
LIN {X 0,Y 183.689,Z 289.124,A -85,B 0,C 180,E1 -23910.367,E2 -23910.367} C_VEL
LIN {X 0,Y 180.855,Z 285.054,A -85,B 0,C 180,E1 -23912.989,E2 -23912.989} C_VEL
LIN {X 0,Y 178.019,Z 281.521,A -85,B 0,C 180,E1 -23916.009,E2 -23916.009} C_VEL
LIN {X 0,Y 177.217,Z 280.206,A -85,B 0,C 180,E1 -23917.022,E2 -23917.022} C_VEL
LIN {X 0,Y 174.637,Z 277.607,A -85,B 0,C 180,E1 -23920.636,E2 -23920.636} C_VEL
LIN {X 0,Y 173.419,Z 275.019,A -85,B 0,C 180,E1 -23923.142,E2 -23923.142} C_VEL
LIN {X 0,Y 170.968,Z 273.108,A -85,B 0,C 180,E1 -23931.728,E2 -23931.728} C_VEL
LIN {X 0,Y 171.725,Z 273.494,A -85,B 0,C 180,E1 -23938.828,E2 -23938.828} C_VEL
LIN {X 0,Y 173.853,Z 275.163,A -85,B 0,C 180,E1 -23944.057,E2 -23944.057} C_VEL
LIN {X 0,Y 175.669,Z 278.51,A -85,B 0,C 180,E1 -23947.324,E2 -23947.324} C_VEL
LIN {X 0,Y 177.617,Z 280.479,A -85,B 0,C 180,E1 -23949.852,E2 -23949.852} C_VEL
LIN {X 0,Y 180.166,Z 284.293,A -85,B 0,C 180,E1 -23952.745,E2 -23952.745} C_VEL
LIN {X 0,Y 181.403,Z 285.722,A -85,B 0,C 180,E1 -23953.942,E2 -23953.942} C_VEL
LIN {X 0,Y 185.016,Z 290.848,A -85,B 0,C 180,E1 -23957.131,E2 -23957.131} C_VEL
LIN {X 0,Y 188.092,Z 295.332,A -85,B 0,C 180,E1 -23959.491,E2 -23959.491} C_VEL
LIN {X 0,Y 192.241,Z 301.565,A -85,B 0,C 180,E1 -23962.304,E2 -23962.304} C_VEL
LIN {X 0,Y 198.192,Z 311.646,A -85,B 0,C 180,E1 -23965.818,E2 -23965.818} C_VEL
LIN {X 0,Y 202.443,Z 319.758,A -85,B 0,C 180,E1 -23968.081,E2 -23968.081} C_VEL
LIN {X 0,Y 200.008,Z 349.594,A -85,B 0,C 180,E1 -23969.033,E2 -23969.033} C_VEL
LIN {X 0,Y 198.074,Z 362.41,A -85,B 0,C 180,E1 -23969.773,E2 -23969.773} C_VEL
LIN {X 0,Y 195.281,Z 374.587,A -85,B 0,C 180,E1 -23970.773,E2 -23970.773} C_VEL
LIN {X 0,Y 191.832,Z 386.188,A -85,B 0,C 180,E1 -23972.095,E2 -23972.095} C_VEL
LIN {X 0,Y 187.367,Z 398.011,A -85,B 0,C 180,E1 -23973.917,E2 -23973.917} C_VEL
LIN {X 0,Y 182.488,Z 408.557,A -85,B 0,C 180,E1 -23976.03,E2 -23976.03} C_VEL
LIN {X 0,Y 177.331,Z 417.939,A -85,B 0,C 180,E1 -23978.493,E2 -23978.493} C_VEL
LIN {X 0,Y 172.469,Z 425.732,A -85,B 0,C 180,E1 -23981.171,E2 -23981.171} C_VEL
LIN {X 0,Y 167.259,Z 433.02,A -85,B 0,C 180,E1 -23984.417,E2 -23984.417} C_VEL
LIN {X 0,Y 162.624,Z 438.905,A -85,B 0,C 180,E1 -23987.948,E2 -23987.948} C_VEL
LIN {X 0,Y 158.54,Z 443.427,A -85,B 0,C 180,E1 -23991.643,E2 -23991.643} C_VEL
LIN {X 0,Y 156.148,Z 445.775,A -85,B 0,C 180,E1 -23994.193,E2 -23994.193} C_VEL
LIN {X 0,Y 154.054,Z 447.671,A -85,B 0,C 180,E1 -23996.812,E2 -23996.812} C_VEL
LIN {X 0,Y 152.299,Z 449.073,A -85,B 0,C 180,E1 -23999.499,E2 -23999.499} C_VEL
LIN {X 0,Y 150.788,Z 450.06,A -85,B 0,C 180,E1 -24002.323,E2 -24002.323} C_VEL
LIN {X 0,Y 149.626,Z 450.589,A -85,B 0,C 180,E1 -24004.996,E2 -24004.996} C_VEL
LIN {X 0,Y 148.71,Z 450.696,A -85,B 0,C 180,E1 -24007.789,E2 -24007.789} C_VEL
LIN {X 0,Y 147.897,Z 450.111,A -85,B 0,C 180,E1 -24011.88,E2 -24011.88} C_VEL
LIN {X 0,Y 147.51,Z 448.504,A -85,B 0,C 180,E1 -24016.222,E2 -24016.222} C_VEL
LIN {X 0,Y 147.707,Z 445.962,A -85,B 0,C 180,E1 -24020.417,E2 -24020.417} C_VEL
LIN {X 0,Y 148.434,Z 442.39,A -85,B 0,C 180,E1 -24024.569,E2 -24024.569} C_VEL
LIN {X 0,Y 149.496,Z 437.713,A -85,B 0,C 180,E1 -24028.656,E2 -24028.656} C_VEL
LIN {X 0,Y 151.015,Z 431.792,A -85,B 0,C 180,E1 -24032.67,E2 -24032.67} C_VEL
LIN {X 0,Y 153.15,Z 424.408,A -85,B 0,C 180,E1 -24036.591,E2 -24036.591} C_VEL
LIN {X 0,Y 155.411,Z 416.858,A -85,B 0,C 180,E1 -24039.766,E2 -24039.766} C_VEL
LIN {X 0,Y 157.994,Z 407.688,A -85,B 0,C 180,E1 -24042.854,E2 -24042.854} C_VEL
LIN {X 0,Y 160.694,Z 397.693,A -85,B 0,C 180,E1 -24045.488,E2 -24045.488} C_VEL
LIN {X 0,Y 163.399,Z 386.217,A -85,B 0,C 180,E1 -24047.848,E2 -24047.848} C_VEL
LIN {X 0,Y 165.466,Z 374.493,A -85,B 0,C 180,E1 -24049.705,E2 -24049.705} C_VEL
LIN {X 0,Y 167.314,Z 362.342,A -85,B 0,C 180,E1 -24051.082,E2 -24051.082} C_VEL
LIN {X 0,Y 168.692,Z 349.261,A -85,B 0,C 180,E1 -24052.096,E2 -24052.096} C_VEL
LIN {X 0,Y 170.516,Z 316.988,A -85,B 0,C 180,E1 -24053.415,E2 -24053.415} C_VEL
LIN {X 0,Y 171.784,Z 291.721,A -85,B 0,C 180,E1 -24054.39,E2 -24054.39} C_VEL
LIN {X 0,Y 167.157,Z 281.274,A -85,B 0,C 180,E1 -24055.951,E2 -24055.951} C_VEL
LIN {X 0,Y 160.668,Z 268.64,A -85,B 0,C 180,E1 -24058.227,E2 -24058.227} C_VEL
LIN {X 0,Y 153.95,Z 257.637,A -85,B 0,C 180,E1 -24060.739,E2 -24060.739} C_VEL
LIN {X 0,Y 152.391,Z 254.994,A -85,B 0,C 180,E1 -24061.373,E2 -24061.373} C_VEL
LIN {X 0,Y 150.743,Z 252.636,A -85,B 0,C 180,E1 -24062.037,E2 -24062.037} C_VEL
LIN {X 0,Y 150.243,Z 250.766,A -85,B 0,C 180,E1 -24062.367,E2 -24062.367} C_VEL
LIN {X 0,Y 150.175,Z 250.77,A -85,B 0,C 180,E1 -24067.476,E2 -24067.476} C_VEL
LIN {X 0,Y 150.138,Z 250.769,A -85,B 0,C 180,E1 -24071.498,E2 -24071.498} C_VEL
LIN {X 0,Y 150.133,Z 250.777,A -85,B 0,C 180,E1 -24075.397,E2 -24075.397} C_VEL
LIN {X 0,Y 150.143,Z 250.768,A -85,B 0,C 180,E1 -24079.055,E2 -24079.055} C_VEL
LIN {X 0,Y 150.182,Z 250.752,A -85,B 0,C 180,E1 -24082.711,E2 -24082.711} C_VEL
LIN {X 0,Y 150.221,Z 250.767,A -85,B 0,C 180,E1 -24087.37,E2 -24087.37} C_VEL
LIN {X 0,Y 150.449,Z 250.708,A -85,B 0,C 180,E1 -24091.044,E2 -24091.044} C_VEL
LIN {X 0,Y 153.786,Z 265.378,A -85,B 0,C 180,E1 -24092.41,E2 -24092.41} C_VEL
LIN {X 0,Y 156.953,Z 278.001,A -85,B 0,C 180,E1 -24093.542,E2 -24093.542} C_VEL
LIN {X 0,Y 153.633,Z 348.648,A -85,B 0,C 180,E1 -24099.847,E2 -24099.847} C_VEL
LIN {X 0,Y 152.866,Z 362.476,A -85,B 0,C 180,E1 -24101.573,E2 -24101.573} C_VEL
LIN {X 0,Y 151.927,Z 376.263,A -85,B 0,C 180,E1 -24103.885,E2 -24103.885} C_VEL
LIN {X 0,Y 151.005,Z 390.063,A -85,B 0,C 180,E1 -24106.886,E2 -24106.886} C_VEL
LIN {X 0,Y 150.185,Z 402.302,A -85,B 0,C 180,E1 -24110.287,E2 -24110.287} C_VEL
LIN {X 0,Y 149.656,Z 412.87,A -85,B 0,C 180,E1 -24113.934,E2 -24113.934} C_VEL
LIN {X 0,Y 149.356,Z 422.328,A -85,B 0,C 180,E1 -24117.977,E2 -24117.977} C_VEL
LIN {X 0,Y 149.237,Z 429.996,A -85,B 0,C 180,E1 -24122.023,E2 -24122.023} C_VEL
LIN {X 0,Y 149.764,Z 437.259,A -85,B 0,C 180,E1 -24126.737,E2 -24126.737} C_VEL
LIN {X 0,Y 151.091,Z 443.265,A -85,B 0,C 180,E1 -24131.651,E2 -24131.651} C_VEL
LIN {X 0,Y 153.165,Z 447.54,A -85,B 0,C 180,E1 -24135.98,E2 -24135.98} C_VEL
LIN {X 0,Y 157.52,Z 451.468,A -85,B 0,C 180,E1 -24140.911,E2 -24140.911} C_VEL
LIN {X 0,Y 163.128,Z 454.057,A -85,B 0,C 180,E1 -24145.52,E2 -24145.52} C_VEL
LIN {X 0,Y 170.423,Z 455.417,A -85,B 0,C 180,E1 -24149.997,E2 -24149.997} C_VEL
LIN {X 0,Y 177.969,Z 455.393,A -85,B 0,C 180,E1 -24153.563,E2 -24153.563} C_VEL
LIN {X 0,Y 186.951,Z 454.101,A -85,B 0,C 180,E1 -24156.976,E2 -24156.976} C_VEL
LIN {X 0,Y 196.856,Z 451.465,A -85,B 0,C 180,E1 -24159.987,E2 -24159.987} C_VEL
LIN {X 0,Y 207.507,Z 447.439,A -85,B 0,C 180,E1 -24162.639,E2 -24162.639} C_VEL
LIN {X 0,Y 208.688,Z 446.929,A -85,B 0,C 180,E1 -24162.907,E2 -24162.907} C_VEL
LIN {X 0,Y 208.854,Z 446.952,A -85,B 0,C 180,E1 -24163.503,E2 -24163.503} C_VEL
LIN {X 0,Y 197.529,Z 452.386,A -85,B 0,C 180,E1 -24166.065,E2 -24166.065} C_VEL
LIN {X 0,Y 189.776,Z 455.437,A -85,B 0,C 180,E1 -24168.192,E2 -24168.192} C_VEL
LIN {X 0,Y 180.209,Z 458.385,A -85,B 0,C 180,E1 -24171.389,E2 -24171.389} C_VEL
LIN {X 0,Y 171.635,Z 460.101,A -85,B 0,C 180,E1 -24175.019,E2 -24175.019} C_VEL
LIN {X 0,Y 164.362,Z 460.643,A -85,B 0,C 180,E1 -24179.126,E2 -24179.126} C_VEL
LIN {X 0,Y 158.491,Z 460.04,A -85,B 0,C 180,E1 -24183.674,E2 -24183.674} C_VEL
LIN {X 0,Y 153.98,Z 458.263,A -85,B 0,C 180,E1 -24188.581,E2 -24188.581} C_VEL
LIN {X 0,Y 152.709,Z 457.225,A -85,B 0,C 180,E1 -24190.616,E2 -24190.616} C_VEL
LIN {X 0,Y 151.001,Z 456.073,A -85,B 0,C 180,E1 -24192.648,E2 -24192.648} C_VEL
LIN {X 0,Y 146.861,Z 454.348,A -85,B 0,C 180,E1 -24195.942,E2 -24195.942} C_VEL
LIN {X 0,Y 143.668,Z 453.99,A -85,B 0,C 180,E1 -24198.661,E2 -24198.661} C_VEL
LIN {X 0,Y 142.071,Z 454.804,A -85,B 0,C 180,E1 -24200.801,E2 -24200.801} C_VEL
LIN {X 0,Y 141.804,Z 455.353,A -85,B 0,C 180,E1 -24201.518,E2 -24201.518} C_VEL
LIN {X 0,Y 141.23,Z 457.787,A -85,B 0,C 180,E1 -24204.413,E2 -24204.413} C_VEL
LIN {X 0,Y 141.156,Z 461.183,A -85,B 0,C 180,E1 -24209.997,E2 -24209.997} C_VEL
LIN {X 0,Y 140.822,Z 462.399,A -85,B 0,C 180,E1 -24213.501,E2 -24213.501} C_VEL
LIN {X 0,Y 140.885,Z 463.11,A -85,B 0,C 180,E1 -24218.604,E2 -24218.604} C_VEL
LIN {X 0,Y 141.361,Z 462.978,A -85,B 0,C 180,E1 -24221.467,E2 -24221.467} C_VEL
LIN {X 0,Y 142.128,Z 462.435,A -85,B 0,C 180,E1 -24224.311,E2 -24224.311} C_VEL
LIN {X 0,Y 144.734,Z 460.154,A -85,B 0,C 180,E1 -24229.868,E2 -24229.868} C_VEL
LIN {X 0,Y 147.632,Z 457.374,A -85,B 0,C 180,E1 -24233.865,E2 -24233.865} C_VEL
LIN {X 0,Y 151.217,Z 453.595,A -85,B 0,C 180,E1 -24237.691,E2 -24237.691} C_VEL
LIN {X 0,Y 155.396,Z 448.712,A -85,B 0,C 180,E1 -24241.336,E2 -24241.336} C_VEL
LIN {X 0,Y 160.357,Z 442.581,A -85,B 0,C 180,E1 -24244.73,E2 -24244.73} C_VEL
LIN {X 0,Y 165.933,Z 434.964,A -85,B 0,C 180,E1 -24247.886,E2 -24247.886} C_VEL
LIN {X 0,Y 170.987,Z 427.184,A -85,B 0,C 180,E1 -24250.339,E2 -24250.339} C_VEL
LIN {X 0,Y 176.847,Z 416.663,A -85,B 0,C 180,E1 -24252.884,E2 -24252.884} C_VEL
LIN {X 0,Y 181.956,Z 405.916,A -85,B 0,C 180,E1 -24254.818,E2 -24254.818} C_VEL
LIN {X 0,Y 186.829,Z 393.675,A -85,B 0,C 180,E1 -24256.393,E2 -24256.393} C_VEL
LIN {X 0,Y 190.544,Z 381.723,A -85,B 0,C 180,E1 -24257.53,E2 -24257.53} C_VEL
LIN {X 0,Y 193.495,Z 368.456,A -85,B 0,C 180,E1 -24258.409,E2 -24258.409} C_VEL
LIN {X 0,Y 195.262,Z 355.447,A -85,B 0,C 180,E1 -24258.989,E2 -24258.989} C_VEL
LIN {X 0,Y 197.595,Z 325.589,A -85,B 0,C 180,E1 -24259.937,E2 -24259.937} C_VEL
LIN {X 0,Y 197.354,Z 321.441,A -85,B 0,C 180,E1 -24260.309,E2 -24260.309} C_VEL
LIN {X 0,Y 192.723,Z 312.863,A -85,B 0,C 180,E1 -24263.035,E2 -24263.035} C_VEL
LIN {X 0,Y 187.503,Z 304.124,A -85,B 0,C 180,E1 -24266.524,E2 -24266.524} C_VEL
LIN {X 0,Y 183.841,Z 298.607,A -85,B 0,C 180,E1 -24269.349,E2 -24269.349} C_VEL
LIN {X 0,Y 181.553,Z 295.226,A -85,B 0,C 180,E1 -24271.34,E2 -24271.34} C_VEL
LIN {X 0,Y 178.845,Z 291.275,A -85,B 0,C 180,E1 -24274.011,E2 -24274.011} C_VEL
LIN {X 0,Y 176.142,Z 287.454,A -85,B 0,C 180,E1 -24277.165,E2 -24277.165} C_VEL
LIN {X 0,Y 173.007,Z 283.666,A -85,B 0,C 180,E1 -24281.956,E2 -24281.956} C_VEL
LIN {X 0,Y 172.204,Z 281.904,A -85,B 0,C 180,E1 -24283.794,E2 -24283.794} C_VEL
LIN {X 0,Y 170.092,Z 280.162,A -85,B 0,C 180,E1 -24291.685,E2 -24291.685} C_VEL
LIN {X 0,Y 170.841,Z 280.545,A -85,B 0,C 180,E1 -24298.822,E2 -24298.822} C_VEL
LIN {X 0,Y 172.726,Z 282.175,A -85,B 0,C 180,E1 -24303.645,E2 -24303.645} C_VEL
LIN {X 0,Y 174.639,Z 285.614,A -85,B 0,C 180,E1 -24307.174,E2 -24307.174} C_VEL
LIN {X 0,Y 176.121,Z 287.173,A -85,B 0,C 180,E1 -24309.185,E2 -24309.185} C_VEL
LIN {X 0,Y 178.667,Z 291.025,A -85,B 0,C 180,E1 -24312.207,E2 -24312.207} C_VEL
LIN {X 0,Y 179.722,Z 292.357,A -85,B 0,C 180,E1 -24313.282,E2 -24313.282} C_VEL
LIN {X 0,Y 183.084,Z 297.298,A -85,B 0,C 180,E1 -24316.398,E2 -24316.398} C_VEL
LIN {X 0,Y 185.749,Z 301.295,A -85,B 0,C 180,E1 -24318.555,E2 -24318.555} C_VEL
LIN {X 0,Y 190.208,Z 308.446,A -85,B 0,C 180,E1 -24321.752,E2 -24321.752} C_VEL
LIN {X 0,Y 195.357,Z 317.422,A -85,B 0,C 180,E1 -24324.935,E2 -24324.935} C_VEL
LIN {X 0,Y 198.123,Z 323.147,A -85,B 0,C 180,E1 -24326.53,E2 -24326.53} C_VEL
LIN {X 0,Y 195.826,Z 349.862,A -85,B 0,C 180,E1 -24327.379,E2 -24327.379} C_VEL
LIN {X 0,Y 193.864,Z 362.503,A -85,B 0,C 180,E1 -24328.105,E2 -24328.105} C_VEL
LIN {X 0,Y 190.991,Z 374.618,A -85,B 0,C 180,E1 -24329.085,E2 -24329.085} C_VEL
LIN {X 0,Y 187.411,Z 386.285,A -85,B 0,C 180,E1 -24330.406,E2 -24330.406} C_VEL
LIN {X 0,Y 182.767,Z 398.166,A -85,B 0,C 180,E1 -24332.228,E2 -24332.228} C_VEL
LIN {X 0,Y 177.688,Z 408.741,A -85,B 0,C 180,E1 -24334.35,E2 -24334.35} C_VEL
LIN {X 0,Y 172.8,Z 417.317,A -85,B 0,C 180,E1 -24336.562,E2 -24336.562} C_VEL
LIN {X 0,Y 167.321,Z 425.805,A -85,B 0,C 180,E1 -24339.476,E2 -24339.476} C_VEL
LIN {X 0,Y 162.144,Z 432.703,A -85,B 0,C 180,E1 -24342.54,E2 -24342.54} C_VEL
LIN {X 0,Y 156.944,Z 438.984,A -85,B 0,C 180,E1 -24346.306,E2 -24346.306} C_VEL
LIN {X 0,Y 152.785,Z 443.385,A -85,B 0,C 180,E1 -24349.914,E2 -24349.914} C_VEL
LIN {X 0,Y 149.87,Z 446.062,A -85,B 0,C 180,E1 -24352.865,E2 -24352.865} C_VEL
LIN {X 0,Y 145.956,Z 449.236,A -85,B 0,C 180,E1 -24358.021,E2 -24358.021} C_VEL
LIN {X 0,Y 144.018,Z 450.404,A -85,B 0,C 180,E1 -24361.451,E2 -24361.451} C_VEL
LIN {X 0,Y 141.909,Z 451.037,A -85,B 0,C 180,E1 -24366.663,E2 -24366.663} C_VEL
LIN {X 0,Y 140.844,Z 450.403,A -85,B 0,C 180,E1 -24371.461,E2 -24371.461} C_VEL
LIN {X 0,Y 140.433,Z 449.013,A -85,B 0,C 180,E1 -24375.512,E2 -24375.512} C_VEL
LIN {X 0,Y 140.453,Z 447.477,A -85,B 0,C 180,E1 -24378.457,E2 -24378.457} C_VEL
LIN {X 0,Y 140.992,Z 444.351,A -85,B 0,C 180,E1 -24382.845,E2 -24382.845} C_VEL
LIN {X 0,Y 141.929,Z 440.163,A -85,B 0,C 180,E1 -24387.165,E2 -24387.165} C_VEL
LIN {X 0,Y 143.61,Z 433.794,A -85,B 0,C 180,E1 -24392.107,E2 -24392.107} C_VEL
LIN {X 0,Y 145.69,Z 426.819,A -85,B 0,C 180,E1 -24396.234,E2 -24396.234} C_VEL
LIN {X 0,Y 148.389,Z 418.082,A -85,B 0,C 180,E1 -24400.233,E2 -24400.233} C_VEL
LIN {X 0,Y 151.077,Z 409.132,A -85,B 0,C 180,E1 -24403.453,E2 -24403.453} C_VEL
LIN {X 0,Y 153.87,Z 399.42,A -85,B 0,C 180,E1 -24406.194,E2 -24406.194} C_VEL
LIN {X 0,Y 156.671,Z 388.249,A -85,B 0,C 180,E1 -24408.643,E2 -24408.643} C_VEL
LIN {X 0,Y 158.754,Z 377.974,A -85,B 0,C 180,E1 -24410.406,E2 -24410.406} C_VEL
LIN {X 0,Y 160.483,Z 367.052,A -85,B 0,C 180,E1 -24411.857,E2 -24411.857} C_VEL
LIN {X 0,Y 162.132,Z 354.414,A -85,B 0,C 180,E1 -24413.021,E2 -24413.021} C_VEL
LIN {X 0,Y 163.215,Z 340.913,A -85,B 0,C 180,E1 -24413.768,E2 -24413.768} C_VEL
LIN {X 0,Y 165.727,Z 293.588,A -85,B 0,C 180,E1 -24415.644,E2 -24415.644} C_VEL
LIN {X 0,Y 161.258,Z 283.551,A -85,B 0,C 180,E1 -24417.255,E2 -24417.255} C_VEL
LIN {X 0,Y 154.673,Z 270.832,A -85,B 0,C 180,E1 -24419.746,E2 -24419.746} C_VEL
LIN {X 0,Y 147.882,Z 259.764,A -85,B 0,C 180,E1 -24422.522,E2 -24422.522} C_VEL
LIN {X 0,Y 145.403,Z 256.018,A -85,B 0,C 180,E1 -24423.612,E2 -24423.612} C_VEL
LIN {X 0,Y 143.584,Z 253.407,A -85,B 0,C 180,E1 -24424.439,E2 -24424.439} C_VEL
LIN {X 0,Y 143.109,Z 251.65,A -85,B 0,C 180,E1 -24424.793,E2 -24424.793} C_VEL
LIN {X 0,Y 143.058,Z 251.665,A -85,B 0,C 180,E1 -24429.695,E2 -24429.695} C_VEL
LIN {X 0,Y 143.039,Z 251.647,A -85,B 0,C 180,E1 -24433.465,E2 -24433.465} C_VEL
LIN {X 0,Y 143.044,Z 251.663,A -85,B 0,C 180,E1 -24437.479,E2 -24437.479} C_VEL
LIN {X 0,Y 143.077,Z 251.632,A -85,B 0,C 180,E1 -24441.811,E2 -24441.811} C_VEL
LIN {X 0,Y 143.188,Z 251.644,A -85,B 0,C 180,E1 -24447.322,E2 -24447.322} C_VEL
LIN {X 0,Y 143.368,Z 251.589,A -85,B 0,C 180,E1 -24450.971,E2 -24450.971} C_VEL
LIN {X 0,Y 146.938,Z 267.248,A -85,B 0,C 180,E1 -24452.499,E2 -24452.499} C_VEL
LIN {X 0,Y 149.758,Z 277.983,A -85,B 0,C 180,E1 -24453.498,E2 -24453.498} C_VEL
LIN {X 0,Y 146.717,Z 345.517,A -85,B 0,C 180,E1 -24459.86,E2 -24459.86} C_VEL
LIN {X 0,Y 145.99,Z 359.652,A -85,B 0,C 180,E1 -24461.583,E2 -24461.583} C_VEL
LIN {X 0,Y 145.128,Z 373.196,A -85,B 0,C 180,E1 -24463.831,E2 -24463.831} C_VEL
LIN {X 0,Y 144.264,Z 385.975,A -85,B 0,C 180,E1 -24466.572,E2 -24466.572} C_VEL
LIN {X 0,Y 143.472,Z 398.004,A -85,B 0,C 180,E1 -24469.828,E2 -24469.828} C_VEL
LIN {X 0,Y 142.978,Z 407.444,A -85,B 0,C 180,E1 -24472.941,E2 -24472.941} C_VEL
LIN {X 0,Y 142.611,Z 416.324,A -85,B 0,C 180,E1 -24476.468,E2 -24476.468} C_VEL
LIN {X 0,Y 142.505,Z 423.743,A -85,B 0,C 180,E1 -24479.999,E2 -24479.999} C_VEL
LIN {X 0,Y 142.549,Z 431.108,A -85,B 0,C 180,E1 -24484.24,E2 -24484.24} C_VEL
LIN {X 0,Y 143.25,Z 437.205,A -85,B 0,C 180,E1 -24488.463,E2 -24488.463} C_VEL
LIN {X 0,Y 145.017,Z 443.692,A -85,B 0,C 180,E1 -24494.023,E2 -24494.023} C_VEL
LIN {X 0,Y 147.466,Z 447.612,A -85,B 0,C 180,E1 -24498.045,E2 -24498.045} C_VEL
LIN {X 0,Y 150.96,Z 450.744,A -85,B 0,C 180,E1 -24501.866,E2 -24501.866} C_VEL
LIN {X 0,Y 156.777,Z 453.802,A -85,B 0,C 180,E1 -24506.633,E2 -24506.633} C_VEL
LIN {X 0,Y 163.853,Z 455.588,A -85,B 0,C 180,E1 -24510.977,E2 -24510.977} C_VEL
LIN {X 0,Y 172.122,Z 456.1,A -85,B 0,C 180,E1 -24514.864,E2 -24514.864} C_VEL
LIN {X 0,Y 181.387,Z 455.35,A -85,B 0,C 180,E1 -24518.311,E2 -24518.311} C_VEL
LIN {X 0,Y 191.589,Z 453.299,A -85,B 0,C 180,E1 -24521.322,E2 -24521.322} C_VEL
LIN {X 0,Y 197.829,Z 451.521,A -85,B 0,C 180,E1 -24522.895,E2 -24522.895} C_VEL
LIN {X 0,Y 196.964,Z 451.947,A -85,B 0,C 180,E1 -24523.578,E2 -24523.578} C_VEL
LIN {X 0,Y 189.814,Z 454.587,A -85,B 0,C 180,E1 -24525.289,E2 -24525.289} C_VEL
LIN {X 0,Y 179.537,Z 457.594,A -85,B 0,C 180,E1 -24528.279,E2 -24528.279} C_VEL
LIN {X 0,Y 170.188,Z 459.405,A -85,B 0,C 180,E1 -24531.722,E2 -24531.722} C_VEL
LIN {X 0,Y 161.907,Z 460.051,A -85,B 0,C 180,E1 -24535.643,E2 -24535.643} C_VEL
LIN {X 0,Y 155.136,Z 459.597,A -85,B 0,C 180,E1 -24540.108,E2 -24540.108} C_VEL
LIN {X 0,Y 149.68,Z 458.008,A -85,B 0,C 180,E1 -24544.999,E2 -24544.999} C_VEL
LIN {X 0,Y 145.868,Z 455.281,A -85,B 0,C 180,E1 -24550.287,E2 -24550.287} C_VEL
LIN {X 0,Y 143.894,Z 451.367,A -85,B 0,C 180,E1 -24555.862,E2 -24555.862} C_VEL
LIN {X 0,Y 143.646,Z 450.517,A -85,B 0,C 180,E1 -24557.098,E2 -24557.098} C_VEL
LIN {X 0,Y 141.804,Z 455.353,A -85,B 0,C 180,E1 -24561.518,E2 -24561.518} C_VEL
LIN {X 0,Y 140.699,Z 457.27,A -85,B 0,C 180,E1 -24563.754,E2 -24563.754} C_VEL
LIN {X 0,Y 138.88,Z 458.817,A -85,B 0,C 180,E1 -24565.987,E2 -24565.987} C_VEL
LIN {X 0,Y 134.976,Z 461.088,A -85,B 0,C 180,E1 -24570.638,E2 -24570.638} C_VEL
LIN {X 0,Y 133.697,Z 462.053,A -85,B 0,C 180,E1 -24573.976,E2 -24573.976} C_VEL
LIN {X 0,Y 133.846,Z 462.777,A -85,B 0,C 180,E1 -24579.06,E2 -24579.06} C_VEL
LIN {X 0,Y 135.22,Z 462.197,A -85,B 0,C 180,E1 -24585.059,E2 -24585.059} C_VEL
LIN {X 0,Y 136.394,Z 461.288,A -85,B 0,C 180,E1 -24588.005,E2 -24588.005} C_VEL
LIN {X 0,Y 140.03,Z 458.305,A -85,B 0,C 180,E1 -24593.669,E2 -24593.669} C_VEL
LIN {X 0,Y 143.644,Z 454.941,A -85,B 0,C 180,E1 -24597.694,E2 -24597.694} C_VEL
LIN {X 0,Y 147.801,Z 450.522,A -85,B 0,C 180,E1 -24601.534,E2 -24601.534} C_VEL
LIN {X 0,Y 153.651,Z 443.849,A -85,B 0,C 180,E1 -24605.671,E2 -24605.671} C_VEL
LIN {X 0,Y 159.393,Z 436.593,A -85,B 0,C 180,E1 -24608.922,E2 -24608.922} C_VEL
LIN {X 0,Y 165.655,Z 427.615,A -85,B 0,C 180,E1 -24611.925,E2 -24611.925} C_VEL
LIN {X 0,Y 171.747,Z 417.254,A -85,B 0,C 180,E1 -24614.485,E2 -24614.485} C_VEL
LIN {X 0,Y 177.014,Z 406.742,A -85,B 0,C 180,E1 -24616.43,E2 -24616.43} C_VEL
LIN {X 0,Y 181.379,Z 396.562,A -85,B 0,C 180,E1 -24617.817,E2 -24617.817} C_VEL
LIN {X 0,Y 185.536,Z 384.402,A -85,B 0,C 180,E1 -24619.041,E2 -24619.041} C_VEL
LIN {X 0,Y 188.839,Z 371.368,A -85,B 0,C 180,E1 -24619.985,E2 -24619.985} C_VEL
LIN {X 0,Y 190.95,Z 358.386,A -85,B 0,C 180,E1 -24620.612,E2 -24620.612} C_VEL
LIN {X 0,Y 193.612,Z 326.618,A -85,B 0,C 180,E1 -24621.642,E2 -24621.642} C_VEL
LIN {X 0,Y 193.401,Z 325.07,A -85,B 0,C 180,E1 -24621.847,E2 -24621.847} C_VEL
LIN {X 0,Y 188.637,Z 316.069,A -85,B 0,C 180,E1 -24624.909,E2 -24624.909} C_VEL
LIN {X 0,Y 184.035,Z 308.392,A -85,B 0,C 180,E1 -24628.316,E2 -24628.316} C_VEL
LIN {X 0,Y 180.197,Z 302.267,A -85,B 0,C 180,E1 -24631.656,E2 -24631.656} C_VEL
LIN {X 0,Y 177.257,Z 297.922,A -85,B 0,C 180,E1 -24634.658,E2 -24634.658} C_VEL
LIN {X 0,Y 174.464,Z 293.789,A -85,B 0,C 180,E1 -24638.133,E2 -24638.133} C_VEL
LIN {X 0,Y 171.944,Z 290.76,A -85,B 0,C 180,E1 -24642.226,E2 -24642.226} C_VEL
LIN {X 0,Y 171.173,Z 288.907,A -85,B 0,C 180,E1 -24644.089,E2 -24644.089} C_VEL
LIN {X 0,Y 169.194,Z 287.167,A -85,B 0,C 180,E1 -24651.994,E2 -24651.994} C_VEL
LIN {X 0,Y 169.957,Z 287.592,A -85,B 0,C 180,E1 -24658.816,E2 -24658.816} C_VEL
LIN {X 0,Y 171.549,Z 289.034,A -85,B 0,C 180,E1 -24663.082,E2 -24663.082} C_VEL
LIN {X 0,Y 173.584,Z 292.667,A -85,B 0,C 180,E1 -24666.977,E2 -24666.977} C_VEL
LIN {X 0,Y 174.755,Z 294.059,A -85,B 0,C 180,E1 -24668.657,E2 -24668.657} C_VEL
LIN {X 0,Y 177.554,Z 298.136,A -85,B 0,C 180,E1 -24672.049,E2 -24672.049} C_VEL
